Fanuc TP program (LS listing): FM152248.ls

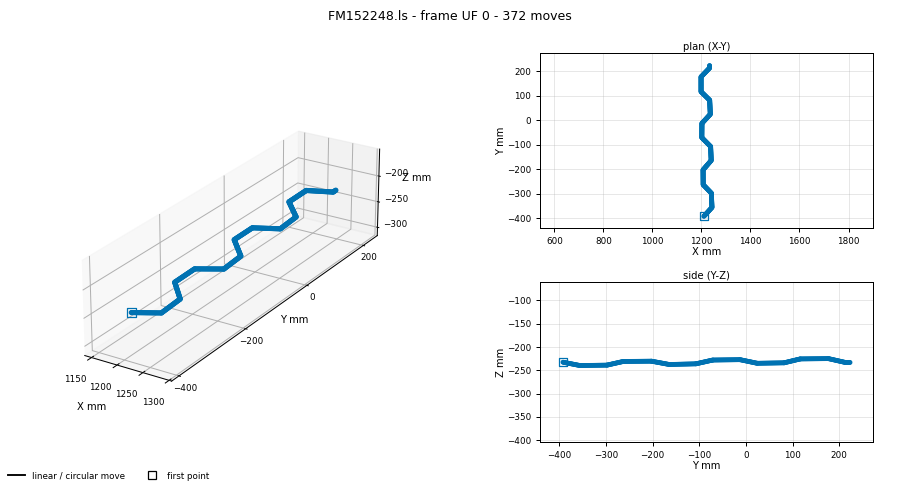
[picture p0: tool path of FM152248.ls in frame UF 0, 372 of 372 moves have a stored position in this frame; points joined in program order, loops and branches not executed]
/PROG  FM152248
/ATTR
OWNER		= MNEDITOR;
COMMENT		= "Auto FANUC move";
PROG_SIZE	= 0;
CREATE		= DATE 26-05-06  TIME 15:22:48;
MODIFIED	= DATE 26-05-06  TIME 15:22:48;
FILE_NAME	= ;
VERSION		= 0;
LINE_COUNT	= 377;
MEMORY_SIZE	= 0;
PROTECT		= READ_WRITE;
TCD:  STACK_SIZE	= 0,
      TASK_PRIORITY	= 50,
      TIME_SLICE	= 0,
      BUSY_LAMP_OFF	= 0,
      ABORT_REQUEST	= 0,
      PAUSE_REQUEST	= 0;
DEFAULT_GROUP	= 1,*,*,*,*;
CONTROL_CODE	= 00000000 00000000;
/MN
   1:  UFRAME_NUM=0 ;
   2:  UTOOL_NUM=1 ;
   3:  R[93]=10 ;
   4:  L P[1] 7mm/sec FINE ;
   5:  L P[2] 7mm/sec CNT50 ;
   6:  L P[3] 7mm/sec CNT50 ;
   7:  L P[4] 7mm/sec CNT50 ;
   8:  L P[5] 7mm/sec CNT50 ;
   9:  L P[6] 7mm/sec CNT50 ;
  10:  L P[7] 7mm/sec CNT50 ;
  11:  L P[8] 7mm/sec CNT50 ;
  12:  L P[9] 7mm/sec CNT50 ;
  13:  L P[10] 7mm/sec CNT50 ;
  14:  L P[11] 7mm/sec CNT50 ;
  15:  L P[12] 7mm/sec CNT50 ;
  16:  L P[13] 7mm/sec CNT50 ;
  17:  L P[14] 7mm/sec CNT50 ;
  18:  L P[15] 7mm/sec CNT50 ;
  19:  L P[16] 7mm/sec CNT50 ;
  20:  L P[17] 7mm/sec CNT50 ;
  21:  L P[18] 7mm/sec CNT50 ;
  22:  L P[19] 7mm/sec CNT50 ;
  23:  L P[20] 7mm/sec CNT50 ;
  24:  L P[21] 7mm/sec CNT50 ;
  25:  L P[22] 7mm/sec CNT50 ;
  26:  L P[23] 7mm/sec CNT50 ;
  27:  L P[24] 7mm/sec CNT50 ;
  28:  L P[25] 7mm/sec CNT50 ;
  29:  L P[26] 7mm/sec CNT50 ;
  30:  L P[27] 7mm/sec CNT50 ;
  31:  L P[28] 7mm/sec CNT50 ;
  32:  L P[29] 7mm/sec CNT50 ;
  33:  L P[30] 7mm/sec CNT50 ;
  34:  L P[31] 7mm/sec CNT50 ;
  35:  L P[32] 7mm/sec CNT50 ;
  36:  L P[33] 7mm/sec CNT50 ;
  37:  L P[34] 7mm/sec CNT50 ;
  38:  L P[35] 7mm/sec CNT50 ;
  39:  L P[36] 7mm/sec CNT50 ;
  40:  L P[37] 7mm/sec CNT50 ;
  41:  L P[38] 7mm/sec CNT50 ;
  42:  L P[39] 7mm/sec CNT50 ;
  43:  L P[40] 7mm/sec CNT50 ;
  44:  L P[41] 7mm/sec CNT50 ;
  45:  L P[42] 7mm/sec CNT50 ;
  46:  L P[43] 7mm/sec CNT50 ;
  47:  L P[44] 7mm/sec CNT50 ;
  48:  L P[45] 7mm/sec CNT50 ;
  49:  L P[46] 7mm/sec CNT50 ;
  50:  L P[47] 7mm/sec CNT50 ;
  51:  L P[48] 7mm/sec CNT50 ;
  52:  L P[49] 7mm/sec CNT50 ;
  53:  L P[50] 7mm/sec CNT50 ;
  54:  L P[51] 7mm/sec CNT50 ;
  55:  L P[52] 7mm/sec CNT50 ;
  56:  L P[53] 7mm/sec CNT50 ;
  57:  L P[54] 7mm/sec CNT50 ;
  58:  L P[55] 7mm/sec CNT50 ;
  59:  L P[56] 7mm/sec CNT50 ;
  60:  L P[57] 7mm/sec CNT50 ;
  61:  L P[58] 7mm/sec CNT50 ;
  62:  L P[59] 7mm/sec CNT50 ;
  63:  L P[60] 7mm/sec CNT50 ;
  64:  L P[61] 7mm/sec CNT50 ;
  65:  L P[62] 7mm/sec CNT50 ;
  66:  L P[63] 7mm/sec CNT50 ;
  67:  L P[64] 7mm/sec CNT50 ;
  68:  L P[65] 7mm/sec CNT50 ;
  69:  L P[66] 7mm/sec CNT50 ;
  70:  L P[67] 7mm/sec CNT50 ;
  71:  L P[68] 7mm/sec CNT50 ;
  72:  L P[69] 7mm/sec CNT50 ;
  73:  L P[70] 7mm/sec CNT50 ;
  74:  L P[71] 7mm/sec CNT50 ;
  75:  L P[72] 7mm/sec CNT50 ;
  76:  L P[73] 7mm/sec CNT50 ;
  77:  L P[74] 7mm/sec CNT50 ;
  78:  L P[75] 7mm/sec CNT50 ;
  79:  L P[76] 7mm/sec CNT50 ;
  80:  L P[77] 7mm/sec CNT50 ;
  81:  L P[78] 7mm/sec CNT50 ;
  82:  L P[79] 7mm/sec CNT50 ;
  83:  L P[80] 7mm/sec CNT50 ;
  84:  L P[81] 7mm/sec CNT50 ;
  85:  L P[82] 7mm/sec CNT50 ;
  86:  L P[83] 7mm/sec CNT50 ;
  87:  L P[84] 7mm/sec CNT50 ;
  88:  L P[85] 7mm/sec CNT50 ;
  89:  L P[86] 7mm/sec CNT50 ;
  90:  L P[87] 7mm/sec CNT50 ;
  91:  L P[88] 7mm/sec CNT50 ;
  92:  L P[89] 7mm/sec CNT50 ;
  93:  L P[90] 7mm/sec CNT50 ;
  94:  L P[91] 7mm/sec CNT50 ;
  95:  L P[92] 7mm/sec CNT50 ;
  96:  L P[93] 7mm/sec CNT50 ;
  97:  L P[94] 7mm/sec CNT50 ;
  98:  L P[95] 7mm/sec CNT50 ;
  99:  L P[96] 7mm/sec CNT50 ;
 100:  L P[97] 7mm/sec CNT50 ;
 101:  L P[98] 7mm/sec CNT50 ;
 102:  L P[99] 7mm/sec CNT50 ;
 103:  L P[100] 7mm/sec CNT50 ;
 104:  L P[101] 7mm/sec CNT50 ;
 105:  L P[102] 7mm/sec CNT50 ;
 106:  L P[103] 7mm/sec CNT50 ;
 107:  L P[104] 7mm/sec CNT50 ;
 108:  L P[105] 7mm/sec CNT50 ;
 109:  L P[106] 7mm/sec CNT50 ;
 110:  L P[107] 7mm/sec CNT50 ;
 111:  L P[108] 7mm/sec CNT50 ;
 112:  L P[109] 7mm/sec CNT50 ;
 113:  L P[110] 7mm/sec CNT50 ;
 114:  L P[111] 7mm/sec CNT50 ;
 115:  L P[112] 7mm/sec CNT50 ;
 116:  L P[113] 7mm/sec CNT50 ;
 117:  L P[114] 7mm/sec CNT50 ;
 118:  L P[115] 7mm/sec CNT50 ;
 119:  L P[116] 7mm/sec CNT50 ;
 120:  L P[117] 7mm/sec CNT50 ;
 121:  L P[118] 7mm/sec CNT50 ;
 122:  L P[119] 7mm/sec CNT50 ;
 123:  L P[120] 7mm/sec CNT50 ;
 124:  L P[121] 7mm/sec CNT50 ;
 125:  L P[122] 7mm/sec CNT50 ;
 126:  L P[123] 7mm/sec CNT50 ;
 127:  L P[124] 7mm/sec CNT50 ;
 128:  L P[125] 7mm/sec CNT50 ;
 129:  L P[126] 7mm/sec CNT50 ;
 130:  L P[127] 7mm/sec CNT50 ;
 131:  L P[128] 7mm/sec CNT50 ;
 132:  L P[129] 7mm/sec CNT50 ;
 133:  L P[130] 7mm/sec CNT50 ;
 134:  L P[131] 7mm/sec CNT50 ;
 135:  L P[132] 7mm/sec CNT50 ;
 136:  L P[133] 7mm/sec CNT50 ;
 137:  L P[134] 7mm/sec CNT50 ;
 138:  L P[135] 7mm/sec CNT50 ;
 139:  L P[136] 7mm/sec CNT50 ;
 140:  L P[137] 7mm/sec CNT50 ;
 141:  L P[138] 7mm/sec CNT50 ;
 142:  L P[139] 7mm/sec CNT50 ;
 143:  L P[140] 7mm/sec CNT50 ;
 144:  L P[141] 7mm/sec CNT50 ;
 145:  L P[142] 7mm/sec CNT50 ;
 146:  L P[143] 7mm/sec CNT50 ;
 147:  L P[144] 7mm/sec CNT50 ;
 148:  L P[145] 7mm/sec CNT50 ;
 149:  L P[146] 7mm/sec CNT50 ;
 150:  L P[147] 7mm/sec CNT50 ;
 151:  L P[148] 7mm/sec CNT50 ;
 152:  L P[149] 7mm/sec CNT50 ;
 153:  L P[150] 7mm/sec CNT50 ;
 154:  L P[151] 7mm/sec CNT50 ;
 155:  L P[152] 7mm/sec CNT50 ;
 156:  L P[153] 7mm/sec CNT50 ;
 157:  L P[154] 7mm/sec CNT50 ;
 158:  L P[155] 7mm/sec CNT50 ;
 159:  L P[156] 7mm/sec CNT50 ;
 160:  L P[157] 7mm/sec CNT50 ;
 161:  L P[158] 7mm/sec CNT50 ;
 162:  L P[159] 7mm/sec CNT50 ;
 163:  L P[160] 7mm/sec CNT50 ;
 164:  L P[161] 7mm/sec CNT50 ;
 165:  L P[162] 7mm/sec CNT50 ;
 166:  L P[163] 7mm/sec CNT50 ;
 167:  L P[164] 7mm/sec CNT50 ;
 168:  L P[165] 7mm/sec CNT50 ;
 169:  L P[166] 7mm/sec CNT50 ;
 170:  L P[167] 7mm/sec CNT50 ;
 171:  L P[168] 7mm/sec CNT50 ;
 172:  L P[169] 7mm/sec CNT50 ;
 173:  L P[170] 7mm/sec CNT50 ;
 174:  L P[171] 7mm/sec CNT50 ;
 175:  L P[172] 7mm/sec CNT50 ;
 176:  L P[173] 7mm/sec CNT50 ;
 177:  L P[174] 7mm/sec CNT50 ;
 178:  L P[175] 7mm/sec CNT50 ;
 179:  L P[176] 7mm/sec CNT50 ;
 180:  L P[177] 7mm/sec CNT50 ;
 181:  L P[178] 7mm/sec CNT50 ;
 182:  L P[179] 7mm/sec CNT50 ;
 183:  L P[180] 7mm/sec CNT50 ;
 184:  L P[181] 7mm/sec CNT50 ;
 185:  L P[182] 7mm/sec CNT50 ;
 186:  L P[183] 7mm/sec CNT50 ;
 187:  L P[184] 7mm/sec CNT50 ;
 188:  L P[185] 7mm/sec CNT50 ;
 189:  L P[186] 7mm/sec CNT50 ;
 190:  L P[187] 7mm/sec CNT50 ;
 191:  L P[188] 7mm/sec CNT50 ;
 192:  L P[189] 7mm/sec CNT50 ;
 193:  L P[190] 7mm/sec CNT50 ;
 194:  L P[191] 7mm/sec CNT50 ;
 195:  L P[192] 7mm/sec CNT50 ;
 196:  L P[193] 7mm/sec CNT50 ;
 197:  L P[194] 7mm/sec CNT50 ;
 198:  L P[195] 7mm/sec CNT50 ;
 199:  L P[196] 7mm/sec CNT50 ;
 200:  L P[197] 7mm/sec CNT50 ;
 201:  L P[198] 7mm/sec CNT50 ;
 202:  L P[199] 7mm/sec CNT50 ;
 203:  L P[200] 7mm/sec CNT50 ;
 204:  L P[201] 7mm/sec CNT50 ;
 205:  L P[202] 7mm/sec CNT50 ;
 206:  L P[203] 7mm/sec CNT50 ;
 207:  L P[204] 7mm/sec CNT50 ;
 208:  L P[205] 7mm/sec CNT50 ;
 209:  L P[206] 7mm/sec CNT50 ;
 210:  L P[207] 7mm/sec CNT50 ;
 211:  L P[208] 7mm/sec CNT50 ;
 212:  L P[209] 7mm/sec CNT50 ;
 213:  L P[210] 7mm/sec CNT50 ;
 214:  L P[211] 7mm/sec CNT50 ;
 215:  L P[212] 7mm/sec CNT50 ;
 216:  L P[213] 7mm/sec CNT50 ;
 217:  L P[214] 7mm/sec CNT50 ;
 218:  L P[215] 7mm/sec CNT50 ;
 219:  L P[216] 7mm/sec CNT50 ;
 220:  L P[217] 7mm/sec CNT50 ;
 221:  L P[218] 7mm/sec CNT50 ;
 222:  L P[219] 7mm/sec CNT50 ;
 223:  L P[220] 7mm/sec CNT50 ;
 224:  L P[221] 7mm/sec CNT50 ;
 225:  L P[222] 7mm/sec CNT50 ;
 226:  L P[223] 7mm/sec CNT50 ;
 227:  L P[224] 7mm/sec CNT50 ;
 228:  L P[225] 7mm/sec CNT50 ;
 229:  L P[226] 7mm/sec CNT50 ;
 230:  L P[227] 7mm/sec CNT50 ;
 231:  L P[228] 7mm/sec CNT50 ;
 232:  L P[229] 7mm/sec CNT50 ;
 233:  L P[230] 7mm/sec CNT50 ;
 234:  L P[231] 7mm/sec CNT50 ;
 235:  L P[232] 7mm/sec CNT50 ;
 236:  L P[233] 7mm/sec CNT50 ;
 237:  L P[234] 7mm/sec CNT50 ;
 238:  L P[235] 7mm/sec CNT50 ;
 239:  L P[236] 7mm/sec CNT50 ;
 240:  L P[237] 7mm/sec CNT50 ;
 241:  L P[238] 7mm/sec CNT50 ;
 242:  L P[239] 7mm/sec CNT50 ;
 243:  L P[240] 7mm/sec CNT50 ;
 244:  L P[241] 7mm/sec CNT50 ;
 245:  L P[242] 7mm/sec CNT50 ;
 246:  L P[243] 7mm/sec CNT50 ;
 247:  L P[244] 7mm/sec CNT50 ;
 248:  L P[245] 7mm/sec CNT50 ;
 249:  L P[246] 7mm/sec CNT50 ;
 250:  L P[247] 7mm/sec CNT50 ;
 251:  L P[248] 7mm/sec CNT50 ;
 252:  L P[249] 7mm/sec CNT50 ;
 253:  L P[250] 7mm/sec CNT50 ;
 254:  L P[251] 7mm/sec CNT50 ;
 255:  L P[252] 7mm/sec CNT50 ;
 256:  L P[253] 7mm/sec CNT50 ;
 257:  L P[254] 7mm/sec CNT50 ;
 258:  L P[255] 7mm/sec CNT50 ;
 259:  L P[256] 7mm/sec CNT50 ;
 260:  L P[257] 7mm/sec CNT50 ;
 261:  L P[258] 7mm/sec CNT50 ;
 262:  L P[259] 7mm/sec CNT50 ;
 263:  L P[260] 7mm/sec CNT50 ;
 264:  L P[261] 7mm/sec CNT50 ;
 265:  L P[262] 7mm/sec CNT50 ;
 266:  L P[263] 7mm/sec CNT50 ;
 267:  L P[264] 7mm/sec CNT50 ;
 268:  L P[265] 7mm/sec CNT50 ;
 269:  L P[266] 7mm/sec CNT50 ;
 270:  L P[267] 7mm/sec CNT50 ;
 271:  L P[268] 7mm/sec CNT50 ;
 272:  L P[269] 7mm/sec CNT50 ;
 273:  L P[270] 7mm/sec CNT50 ;
 274:  L P[271] 7mm/sec CNT50 ;
 275:  L P[272] 7mm/sec CNT50 ;
 276:  L P[273] 7mm/sec CNT50 ;
 277:  L P[274] 7mm/sec CNT50 ;
 278:  L P[275] 7mm/sec CNT50 ;
 279:  L P[276] 7mm/sec CNT50 ;
 280:  L P[277] 7mm/sec CNT50 ;
 281:  L P[278] 7mm/sec CNT50 ;
 282:  L P[279] 7mm/sec CNT50 ;
 283:  L P[280] 7mm/sec CNT50 ;
 284:  L P[281] 7mm/sec CNT50 ;
 285:  L P[282] 7mm/sec CNT50 ;
 286:  L P[283] 7mm/sec CNT50 ;
 287:  L P[284] 7mm/sec CNT50 ;
 288:  L P[285] 7mm/sec CNT50 ;
 289:  L P[286] 7mm/sec CNT50 ;
 290:  L P[287] 7mm/sec CNT50 ;
 291:  L P[288] 7mm/sec CNT50 ;
 292:  L P[289] 7mm/sec CNT50 ;
 293:  L P[290] 7mm/sec CNT50 ;
 294:  L P[291] 7mm/sec CNT50 ;
 295:  L P[292] 7mm/sec CNT50 ;
 296:  L P[293] 7mm/sec CNT50 ;
 297:  L P[294] 7mm/sec CNT50 ;
 298:  L P[295] 7mm/sec CNT50 ;
 299:  L P[296] 7mm/sec CNT50 ;
 300:  L P[297] 7mm/sec CNT50 ;
 301:  L P[298] 7mm/sec CNT50 ;
 302:  L P[299] 7mm/sec CNT50 ;
 303:  L P[300] 7mm/sec CNT50 ;
 304:  L P[301] 7mm/sec CNT50 ;
 305:  L P[302] 7mm/sec CNT50 ;
 306:  L P[303] 7mm/sec CNT50 ;
 307:  L P[304] 7mm/sec CNT50 ;
 308:  L P[305] 7mm/sec CNT50 ;
 309:  L P[306] 7mm/sec CNT50 ;
 310:  L P[307] 7mm/sec CNT50 ;
 311:  L P[308] 7mm/sec CNT50 ;
 312:  L P[309] 7mm/sec CNT50 ;
 313:  L P[310] 7mm/sec CNT50 ;
 314:  L P[311] 7mm/sec CNT50 ;
 315:  L P[312] 7mm/sec CNT50 ;
 316:  L P[313] 7mm/sec CNT50 ;
 317:  L P[314] 7mm/sec CNT50 ;
 318:  L P[315] 7mm/sec CNT50 ;
 319:  L P[316] 7mm/sec CNT50 ;
 320:  L P[317] 7mm/sec CNT50 ;
 321:  L P[318] 7mm/sec CNT50 ;
 322:  L P[319] 7mm/sec CNT50 ;
 323:  L P[320] 7mm/sec CNT50 ;
 324:  L P[321] 7mm/sec CNT50 ;
 325:  L P[322] 7mm/sec CNT50 ;
 326:  L P[323] 7mm/sec CNT50 ;
 327:  L P[324] 7mm/sec CNT50 ;
 328:  L P[325] 7mm/sec CNT50 ;
 329:  L P[326] 7mm/sec CNT50 ;
 330:  L P[327] 7mm/sec CNT50 ;
 331:  L P[328] 7mm/sec CNT50 ;
 332:  L P[329] 7mm/sec CNT50 ;
 333:  L P[330] 7mm/sec CNT50 ;
 334:  L P[331] 7mm/sec CNT50 ;
 335:  L P[332] 7mm/sec CNT50 ;
 336:  L P[333] 7mm/sec CNT50 ;
 337:  L P[334] 7mm/sec CNT50 ;
 338:  L P[335] 7mm/sec CNT50 ;
 339:  L P[336] 7mm/sec CNT50 ;
 340:  L P[337] 7mm/sec CNT50 ;
 341:  L P[338] 7mm/sec CNT50 ;
 342:  L P[339] 7mm/sec CNT50 ;
 343:  L P[340] 7mm/sec CNT50 ;
 344:  L P[341] 7mm/sec CNT50 ;
 345:  L P[342] 7mm/sec CNT50 ;
 346:  L P[343] 7mm/sec CNT50 ;
 347:  L P[344] 7mm/sec CNT50 ;
 348:  L P[345] 7mm/sec CNT50 ;
 349:  L P[346] 7mm/sec CNT50 ;
 350:  L P[347] 7mm/sec CNT50 ;
 351:  L P[348] 7mm/sec CNT50 ;
 352:  L P[349] 7mm/sec CNT50 ;
 353:  L P[350] 7mm/sec CNT50 ;
 354:  L P[351] 7mm/sec CNT50 ;
 355:  L P[352] 7mm/sec CNT50 ;
 356:  L P[353] 7mm/sec CNT50 ;
 357:  L P[354] 7mm/sec CNT50 ;
 358:  L P[355] 7mm/sec CNT50 ;
 359:  L P[356] 7mm/sec CNT50 ;
 360:  L P[357] 7mm/sec CNT50 ;
 361:  L P[358] 7mm/sec CNT50 ;
 362:  L P[359] 7mm/sec CNT50 ;
 363:  L P[360] 7mm/sec CNT50 ;
 364:  L P[361] 7mm/sec CNT50 ;
 365:  L P[362] 7mm/sec CNT50 ;
 366:  L P[363] 7mm/sec CNT50 ;
 367:  L P[364] 7mm/sec CNT50 ;
 368:  L P[365] 7mm/sec CNT50 ;
 369:  L P[366] 7mm/sec CNT50 ;
 370:  L P[367] 7mm/sec CNT50 ;
 371:  L P[368] 7mm/sec CNT50 ;
 372:  L P[369] 7mm/sec CNT50 ;
 373:  L P[370] 7mm/sec CNT50 ;
 374:  L P[371] 7mm/sec CNT50 ;
 375:  L P[372] 7mm/sec FINE ;
 376:  R[93]=1 ;
 377:  END ;
/POS
P[1]{
   GP1:
	UF : 0, UT : 1,		CONFIG : 'N U T, 0, 0, 0',
	X = 1209.863  mm,	Y = -392.091  mm,	Z = -232.573  mm,
	W = 0.000 deg,	P = 30.000 deg,	R = 160.000 deg
};
P[2]{
   GP1:
	UF : 0, UT : 1,		CONFIG : 'N U T, 0, 0, 0',
	X = 1211.194  mm,	Y = -390.625  mm,	Z = -232.860  mm,
	W = 0.000 deg,	P = 30.000 deg,	R = 160.000 deg
};
P[3]{
   GP1:
	UF : 0, UT : 1,		CONFIG : 'N U T, 0, 0, 0',
	X = 1212.524  mm,	Y = -389.159  mm,	Z = -233.146  mm,
	W = 0.000 deg,	P = 30.000 deg,	R = 160.000 deg
};
P[4]{
   GP1:
	UF : 0, UT : 1,		CONFIG : 'N U T, 0, 0, 0',
	X = 1213.854  mm,	Y = -387.693  mm,	Z = -233.432  mm,
	W = 0.000 deg,	P = 30.000 deg,	R = 160.000 deg
};
P[5]{
   GP1:
	UF : 0, UT : 1,		CONFIG : 'N U T, 0, 0, 0',
	X = 1215.184  mm,	Y = -386.228  mm,	Z = -233.719  mm,
	W = 0.000 deg,	P = 30.000 deg,	R = 160.000 deg
};
P[6]{
   GP1:
	UF : 0, UT : 1,		CONFIG : 'N U T, 0, 0, 0',
	X = 1216.515  mm,	Y = -384.762  mm,	Z = -234.005  mm,
	W = 0.000 deg,	P = 30.000 deg,	R = 160.000 deg
};
P[7]{
   GP1:
	UF : 0, UT : 1,		CONFIG : 'N U T, 0, 0, 0',
	X = 1217.845  mm,	Y = -383.296  mm,	Z = -234.291  mm,
	W = 0.000 deg,	P = 30.000 deg,	R = 160.000 deg
};
P[8]{
   GP1:
	UF : 0, UT : 1,		CONFIG : 'N U T, 0, 0, 0',
	X = 1219.175  mm,	Y = -381.830  mm,	Z = -234.578  mm,
	W = 0.000 deg,	P = 30.000 deg,	R = 160.000 deg
};
P[9]{
   GP1:
	UF : 0, UT : 1,		CONFIG : 'N U T, 0, 0, 0',
	X = 1220.505  mm,	Y = -380.365  mm,	Z = -234.864  mm,
	W = 0.000 deg,	P = 30.000 deg,	R = 160.000 deg
};
P[10]{
   GP1:
	UF : 0, UT : 1,		CONFIG : 'N U T, 0, 0, 0',
	X = 1221.836  mm,	Y = -378.899  mm,	Z = -235.150  mm,
	W = 0.000 deg,	P = 30.000 deg,	R = 160.000 deg
};
P[11]{
   GP1:
	UF : 0, UT : 1,		CONFIG : 'N U T, 0, 0, 0',
	X = 1223.166  mm,	Y = -377.433  mm,	Z = -235.437  mm,
	W = 0.000 deg,	P = 30.000 deg,	R = 160.000 deg
};
P[12]{
   GP1:
	UF : 0, UT : 1,		CONFIG : 'N U T, 0, 0, 0',
	X = 1224.496  mm,	Y = -375.967  mm,	Z = -235.723  mm,
	W = 0.000 deg,	P = 30.000 deg,	R = 160.000 deg
};
P[13]{
   GP1:
	UF : 0, UT : 1,		CONFIG : 'N U T, 0, 0, 0',
	X = 1225.826  mm,	Y = -374.502  mm,	Z = -236.010  mm,
	W = 0.000 deg,	P = 30.000 deg,	R = 160.000 deg
};
P[14]{
   GP1:
	UF : 0, UT : 1,		CONFIG : 'N U T, 0, 0, 0',
	X = 1227.157  mm,	Y = -373.036  mm,	Z = -236.296  mm,
	W = 0.000 deg,	P = 30.000 deg,	R = 160.000 deg
};
P[15]{
   GP1:
	UF : 0, UT : 1,		CONFIG : 'N U T, 0, 0, 0',
	X = 1228.487  mm,	Y = -371.570  mm,	Z = -236.582  mm,
	W = 0.000 deg,	P = 30.000 deg,	R = 160.000 deg
};
P[16]{
   GP1:
	UF : 0, UT : 1,		CONFIG : 'N U T, 0, 0, 0',
	X = 1229.817  mm,	Y = -370.104  mm,	Z = -236.869  mm,
	W = 0.000 deg,	P = 30.000 deg,	R = 160.000 deg
};
P[17]{
   GP1:
	UF : 0, UT : 1,		CONFIG : 'N U T, 0, 0, 0',
	X = 1231.147  mm,	Y = -368.639  mm,	Z = -237.155  mm,
	W = 0.000 deg,	P = 30.000 deg,	R = 160.000 deg
};
P[18]{
   GP1:
	UF : 0, UT : 1,		CONFIG : 'N U T, 0, 0, 0',
	X = 1232.478  mm,	Y = -367.173  mm,	Z = -237.441  mm,
	W = 0.000 deg,	P = 30.000 deg,	R = 160.000 deg
};
P[19]{
   GP1:
	UF : 0, UT : 1,		CONFIG : 'N U T, 0, 0, 0',
	X = 1233.808  mm,	Y = -365.707  mm,	Z = -237.728  mm,
	W = 0.000 deg,	P = 30.000 deg,	R = 160.000 deg
};
P[20]{
   GP1:
	UF : 0, UT : 1,		CONFIG : 'N U T, 0, 0, 0',
	X = 1235.138  mm,	Y = -364.241  mm,	Z = -238.014  mm,
	W = 0.000 deg,	P = 30.000 deg,	R = 160.000 deg
};
P[21]{
   GP1:
	UF : 0, UT : 1,		CONFIG : 'N U T, 0, 0, 0',
	X = 1236.468  mm,	Y = -362.776  mm,	Z = -238.300  mm,
	W = 0.000 deg,	P = 30.000 deg,	R = 164.441 deg
};
P[22]{
   GP1:
	UF : 0, UT : 1,		CONFIG : 'N U T, 0, 0, 0',
	X = 1237.799  mm,	Y = -361.310  mm,	Z = -238.587  mm,
	W = 0.000 deg,	P = 30.000 deg,	R = 168.883 deg
};
P[23]{
   GP1:
	UF : 0, UT : 1,		CONFIG : 'N U T, 0, 0, 0',
	X = 1239.129  mm,	Y = -359.844  mm,	Z = -238.873  mm,
	W = 0.000 deg,	P = 30.000 deg,	R = 173.324 deg
};
P[24]{
   GP1:
	UF : 0, UT : 1,		CONFIG : 'N U T, 0, 0, 0',
	X = 1240.459  mm,	Y = -358.378  mm,	Z = -239.159  mm,
	W = 0.000 deg,	P = 30.000 deg,	R = 177.765 deg
};
P[25]{
   GP1:
	UF : 0, UT : 1,		CONFIG : 'N U T, 0, 0, 0',
	X = 1241.789  mm,	Y = -356.912  mm,	Z = -239.446  mm,
	W = 0.000 deg,	P = 30.000 deg,	R = -177.793 deg
};
P[26]{
   GP1:
	UF : 0, UT : 1,		CONFIG : 'N U T, 0, 0, 0',
	X = 1242.946  mm,	Y = -355.638  mm,	Z = -239.695  mm,
	W = 0.000 deg,	P = 30.000 deg,	R = -177.793 deg
};
P[27]{
   GP1:
	UF : 0, UT : 1,		CONFIG : 'N U T, 0, 0, 0',
	X = 1242.936  mm,	Y = -355.377  mm,	Z = -239.691  mm,
	W = 0.000 deg,	P = 30.000 deg,	R = -177.793 deg
};
P[28]{
   GP1:
	UF : 0, UT : 1,		CONFIG : 'N U T, 0, 0, 0',
	X = 1242.859  mm,	Y = -353.379  mm,	Z = -239.662  mm,
	W = 0.000 deg,	P = 30.000 deg,	R = -177.793 deg
};
P[29]{
   GP1:
	UF : 0, UT : 1,		CONFIG : 'N U T, 0, 0, 0',
	X = 1242.782  mm,	Y = -351.381  mm,	Z = -239.633  mm,
	W = 0.000 deg,	P = 30.000 deg,	R = -177.793 deg
};
P[30]{
   GP1:
	UF : 0, UT : 1,		CONFIG : 'N U T, 0, 0, 0',
	X = 1242.705  mm,	Y = -349.382  mm,	Z = -239.604  mm,
	W = 0.000 deg,	P = 30.000 deg,	R = -177.793 deg
};
P[31]{
   GP1:
	UF : 0, UT : 1,		CONFIG : 'N U T, 0, 0, 0',
	X = 1242.628  mm,	Y = -347.384  mm,	Z = -239.575  mm,
	W = 0.000 deg,	P = 30.000 deg,	R = -177.793 deg
};
P[32]{
   GP1:
	UF : 0, UT : 1,		CONFIG : 'N U T, 0, 0, 0',
	X = 1242.551  mm,	Y = -345.386  mm,	Z = -239.546  mm,
	W = 0.000 deg,	P = 30.000 deg,	R = -177.793 deg
};
P[33]{
   GP1:
	UF : 0, UT : 1,		CONFIG : 'N U T, 0, 0, 0',
	X = 1242.474  mm,	Y = -343.388  mm,	Z = -239.517  mm,
	W = 0.000 deg,	P = 30.000 deg,	R = -177.793 deg
};
P[34]{
   GP1:
	UF : 0, UT : 1,		CONFIG : 'N U T, 0, 0, 0',
	X = 1242.397  mm,	Y = -341.389  mm,	Z = -239.488  mm,
	W = 0.000 deg,	P = 30.000 deg,	R = -177.793 deg
};
P[35]{
   GP1:
	UF : 0, UT : 1,		CONFIG : 'N U T, 0, 0, 0',
	X = 1242.320  mm,	Y = -339.391  mm,	Z = -239.459  mm,
	W = 0.000 deg,	P = 30.000 deg,	R = -177.793 deg
};
P[36]{
   GP1:
	UF : 0, UT : 1,		CONFIG : 'N U T, 0, 0, 0',
	X = 1242.243  mm,	Y = -337.393  mm,	Z = -239.430  mm,
	W = 0.000 deg,	P = 30.000 deg,	R = -177.793 deg
};
P[37]{
   GP1:
	UF : 0, UT : 1,		CONFIG : 'N U T, 0, 0, 0',
	X = 1242.166  mm,	Y = -335.394  mm,	Z = -239.401  mm,
	W = 0.000 deg,	P = 30.000 deg,	R = -177.793 deg
};
P[38]{
   GP1:
	UF : 0, UT : 1,		CONFIG : 'N U T, 0, 0, 0',
	X = 1242.089  mm,	Y = -333.396  mm,	Z = -239.372  mm,
	W = 0.000 deg,	P = 30.000 deg,	R = -177.793 deg
};
P[39]{
   GP1:
	UF : 0, UT : 1,		CONFIG : 'N U T, 0, 0, 0',
	X = 1242.012  mm,	Y = -331.398  mm,	Z = -239.342  mm,
	W = 0.000 deg,	P = 30.000 deg,	R = -177.793 deg
};
P[40]{
   GP1:
	UF : 0, UT : 1,		CONFIG : 'N U T, 0, 0, 0',
	X = 1241.935  mm,	Y = -329.399  mm,	Z = -239.313  mm,
	W = 0.000 deg,	P = 30.000 deg,	R = -177.793 deg
};
P[41]{
   GP1:
	UF : 0, UT : 1,		CONFIG : 'N U T, 0, 0, 0',
	X = 1241.858  mm,	Y = -327.401  mm,	Z = -239.284  mm,
	W = 0.000 deg,	P = 30.000 deg,	R = -177.793 deg
};
P[42]{
   GP1:
	UF : 0, UT : 1,		CONFIG : 'N U T, 0, 0, 0',
	X = 1241.781  mm,	Y = -325.403  mm,	Z = -239.255  mm,
	W = 0.000 deg,	P = 30.000 deg,	R = -177.793 deg
};
P[43]{
   GP1:
	UF : 0, UT : 1,		CONFIG : 'N U T, 0, 0, 0',
	X = 1241.704  mm,	Y = -323.405  mm,	Z = -239.226  mm,
	W = 0.000 deg,	P = 30.000 deg,	R = -177.793 deg
};
P[44]{
   GP1:
	UF : 0, UT : 1,		CONFIG : 'N U T, 0, 0, 0',
	X = 1241.627  mm,	Y = -321.406  mm,	Z = -239.197  mm,
	W = 0.000 deg,	P = 30.000 deg,	R = -177.793 deg
};
P[45]{
   GP1:
	UF : 0, UT : 1,		CONFIG : 'N U T, 0, 0, 0',
	X = 1241.550  mm,	Y = -319.408  mm,	Z = -239.168  mm,
	W = 0.000 deg,	P = 30.000 deg,	R = -177.793 deg
};
P[46]{
   GP1:
	UF : 0, UT : 1,		CONFIG : 'N U T, 0, 0, 0',
	X = 1241.473  mm,	Y = -317.410  mm,	Z = -239.139  mm,
	W = 0.000 deg,	P = 30.000 deg,	R = -177.793 deg
};
P[47]{
   GP1:
	UF : 0, UT : 1,		CONFIG : 'N U T, 0, 0, 0',
	X = 1241.396  mm,	Y = -315.411  mm,	Z = -239.110  mm,
	W = 0.000 deg,	P = 30.000 deg,	R = -177.793 deg
};
P[48]{
   GP1:
	UF : 0, UT : 1,		CONFIG : 'N U T, 0, 0, 0',
	X = 1241.319  mm,	Y = -313.413  mm,	Z = -239.081  mm,
	W = 0.000 deg,	P = 30.000 deg,	R = -177.793 deg
};
P[49]{
   GP1:
	UF : 0, UT : 1,		CONFIG : 'N U T, 0, 0, 0',
	X = 1241.242  mm,	Y = -311.415  mm,	Z = -239.052  mm,
	W = 0.000 deg,	P = 30.000 deg,	R = -177.793 deg
};
P[50]{
   GP1:
	UF : 0, UT : 1,		CONFIG : 'N U T, 0, 0, 0',
	X = 1241.165  mm,	Y = -309.416  mm,	Z = -239.023  mm,
	W = 0.000 deg,	P = 30.000 deg,	R = -177.330 deg
};
P[51]{
   GP1:
	UF : 0, UT : 1,		CONFIG : 'N U T, 0, 0, 0',
	X = 1241.088  mm,	Y = -307.418  mm,	Z = -238.994  mm,
	W = 0.000 deg,	P = 30.000 deg,	R = -173.771 deg
};
P[52]{
   GP1:
	UF : 0, UT : 1,		CONFIG : 'N U T, 0, 0, 0',
	X = 1241.011  mm,	Y = -305.420  mm,	Z = -238.965  mm,
	W = 0.000 deg,	P = 30.000 deg,	R = -170.213 deg
};
P[53]{
   GP1:
	UF : 0, UT : 1,		CONFIG : 'N U T, 0, 0, 0',
	X = 1240.934  mm,	Y = -303.421  mm,	Z = -238.936  mm,
	W = 0.000 deg,	P = 30.000 deg,	R = -166.654 deg
};
P[54]{
   GP1:
	UF : 0, UT : 1,		CONFIG : 'N U T, 0, 0, 0',
	X = 1240.857  mm,	Y = -301.423  mm,	Z = -238.907  mm,
	W = 0.000 deg,	P = 30.000 deg,	R = -163.095 deg
};
P[55]{
   GP1:
	UF : 0, UT : 1,		CONFIG : 'N U T, 0, 0, 0',
	X = 1240.780  mm,	Y = -299.425  mm,	Z = -238.878  mm,
	W = 0.000 deg,	P = 30.000 deg,	R = -160.000 deg
};
P[56]{
   GP1:
	UF : 0, UT : 1,		CONFIG : 'N U T, 0, 0, 0',
	X = 1240.717  mm,	Y = -297.777  mm,	Z = -238.854  mm,
	W = 0.000 deg,	P = 30.000 deg,	R = -160.000 deg
};
P[57]{
   GP1:
	UF : 0, UT : 1,		CONFIG : 'N U T, 0, 0, 0',
	X = 1240.477  mm,	Y = -297.528  mm,	Z = -238.798  mm,
	W = 0.000 deg,	P = 30.000 deg,	R = -160.000 deg
};
P[58]{
   GP1:
	UF : 0, UT : 1,		CONFIG : 'N U T, 0, 0, 0',
	X = 1239.108  mm,	Y = -296.105  mm,	Z = -238.477  mm,
	W = 0.000 deg,	P = 30.000 deg,	R = -160.000 deg
};
P[59]{
   GP1:
	UF : 0, UT : 1,		CONFIG : 'N U T, 0, 0, 0',
	X = 1237.740  mm,	Y = -294.682  mm,	Z = -238.157  mm,
	W = 0.000 deg,	P = 30.000 deg,	R = -160.000 deg
};
P[60]{
   GP1:
	UF : 0, UT : 1,		CONFIG : 'N U T, 0, 0, 0',
	X = 1236.371  mm,	Y = -293.259  mm,	Z = -237.836  mm,
	W = 0.000 deg,	P = 30.000 deg,	R = -160.000 deg
};
P[61]{
   GP1:
	UF : 0, UT : 1,		CONFIG : 'N U T, 0, 0, 0',
	X = 1235.003  mm,	Y = -291.836  mm,	Z = -237.516  mm,
	W = 0.000 deg,	P = 30.000 deg,	R = -160.000 deg
};
P[62]{
   GP1:
	UF : 0, UT : 1,		CONFIG : 'N U T, 0, 0, 0',
	X = 1233.634  mm,	Y = -290.413  mm,	Z = -237.196  mm,
	W = 0.000 deg,	P = 30.000 deg,	R = -160.000 deg
};
P[63]{
   GP1:
	UF : 0, UT : 1,		CONFIG : 'N U T, 0, 0, 0',
	X = 1232.265  mm,	Y = -288.990  mm,	Z = -236.875  mm,
	W = 0.000 deg,	P = 30.000 deg,	R = -160.000 deg
};
P[64]{
   GP1:
	UF : 0, UT : 1,		CONFIG : 'N U T, 0, 0, 0',
	X = 1230.897  mm,	Y = -287.568  mm,	Z = -236.555  mm,
	W = 0.000 deg,	P = 30.000 deg,	R = -160.000 deg
};
P[65]{
   GP1:
	UF : 0, UT : 1,		CONFIG : 'N U T, 0, 0, 0',
	X = 1229.528  mm,	Y = -286.145  mm,	Z = -236.234  mm,
	W = 0.000 deg,	P = 30.000 deg,	R = -160.000 deg
};
P[66]{
   GP1:
	UF : 0, UT : 1,		CONFIG : 'N U T, 0, 0, 0',
	X = 1228.160  mm,	Y = -284.722  mm,	Z = -235.914  mm,
	W = 0.000 deg,	P = 30.000 deg,	R = -160.000 deg
};
P[67]{
   GP1:
	UF : 0, UT : 1,		CONFIG : 'N U T, 0, 0, 0',
	X = 1226.791  mm,	Y = -283.299  mm,	Z = -235.594  mm,
	W = 0.000 deg,	P = 30.000 deg,	R = -160.000 deg
};
P[68]{
   GP1:
	UF : 0, UT : 1,		CONFIG : 'N U T, 0, 0, 0',
	X = 1225.423  mm,	Y = -281.876  mm,	Z = -235.273  mm,
	W = 0.000 deg,	P = 30.000 deg,	R = -160.000 deg
};
P[69]{
   GP1:
	UF : 0, UT : 1,		CONFIG : 'N U T, 0, 0, 0',
	X = 1224.054  mm,	Y = -280.453  mm,	Z = -234.953  mm,
	W = 0.000 deg,	P = 30.000 deg,	R = -160.000 deg
};
P[70]{
   GP1:
	UF : 0, UT : 1,		CONFIG : 'N U T, 0, 0, 0',
	X = 1222.686  mm,	Y = -279.031  mm,	Z = -234.632  mm,
	W = 0.000 deg,	P = 30.000 deg,	R = -160.000 deg
};
P[71]{
   GP1:
	UF : 0, UT : 1,		CONFIG : 'N U T, 0, 0, 0',
	X = 1221.317  mm,	Y = -277.608  mm,	Z = -234.312  mm,
	W = 0.000 deg,	P = 30.000 deg,	R = -160.000 deg
};
P[72]{
   GP1:
	UF : 0, UT : 1,		CONFIG : 'N U T, 0, 0, 0',
	X = 1219.949  mm,	Y = -276.185  mm,	Z = -233.992  mm,
	W = 0.000 deg,	P = 30.000 deg,	R = -160.000 deg
};
P[73]{
   GP1:
	UF : 0, UT : 1,		CONFIG : 'N U T, 0, 0, 0',
	X = 1218.580  mm,	Y = -274.762  mm,	Z = -233.671  mm,
	W = 0.000 deg,	P = 30.000 deg,	R = -160.000 deg
};
P[74]{
   GP1:
	UF : 0, UT : 1,		CONFIG : 'N U T, 0, 0, 0',
	X = 1217.212  mm,	Y = -273.339  mm,	Z = -233.351  mm,
	W = 0.000 deg,	P = 30.000 deg,	R = -160.000 deg
};
P[75]{
   GP1:
	UF : 0, UT : 1,		CONFIG : 'N U T, 0, 0, 0',
	X = 1215.843  mm,	Y = -271.916  mm,	Z = -233.030  mm,
	W = 0.000 deg,	P = 30.000 deg,	R = -160.000 deg
};
P[76]{
   GP1:
	UF : 0, UT : 1,		CONFIG : 'N U T, 0, 0, 0',
	X = 1214.475  mm,	Y = -270.494  mm,	Z = -232.710  mm,
	W = 0.000 deg,	P = 30.000 deg,	R = -160.688 deg
};
P[77]{
   GP1:
	UF : 0, UT : 1,		CONFIG : 'N U T, 0, 0, 0',
	X = 1213.106  mm,	Y = -269.071  mm,	Z = -232.390  mm,
	W = 0.000 deg,	P = 30.000 deg,	R = -164.612 deg
};
P[78]{
   GP1:
	UF : 0, UT : 1,		CONFIG : 'N U T, 0, 0, 0',
	X = 1211.738  mm,	Y = -267.648  mm,	Z = -232.069  mm,
	W = 0.000 deg,	P = 30.000 deg,	R = -168.535 deg
};
P[79]{
   GP1:
	UF : 0, UT : 1,		CONFIG : 'N U T, 0, 0, 0',
	X = 1210.369  mm,	Y = -266.225  mm,	Z = -231.749  mm,
	W = 0.000 deg,	P = 30.000 deg,	R = -172.458 deg
};
P[80]{
   GP1:
	UF : 0, UT : 1,		CONFIG : 'N U T, 0, 0, 0',
	X = 1209.000  mm,	Y = -264.802  mm,	Z = -231.429  mm,
	W = 0.000 deg,	P = 30.000 deg,	R = -176.382 deg
};
P[81]{
   GP1:
	UF : 0, UT : 1,		CONFIG : 'N U T, 0, 0, 0',
	X = 1207.632  mm,	Y = -263.379  mm,	Z = -231.108  mm,
	W = 0.000 deg,	P = 30.000 deg,	R = -179.617 deg
};
P[82]{
   GP1:
	UF : 0, UT : 1,		CONFIG : 'N U T, 0, 0, 0',
	X = 1207.094  mm,	Y = -262.820  mm,	Z = -230.982  mm,
	W = 0.000 deg,	P = 30.000 deg,	R = -179.617 deg
};
P[83]{
   GP1:
	UF : 0, UT : 1,		CONFIG : 'N U T, 0, 0, 0',
	X = 1207.086  mm,	Y = -261.606  mm,	Z = -230.970  mm,
	W = 0.000 deg,	P = 30.000 deg,	R = -179.617 deg
};
P[84]{
   GP1:
	UF : 0, UT : 1,		CONFIG : 'N U T, 0, 0, 0',
	X = 1207.073  mm,	Y = -259.606  mm,	Z = -230.950  mm,
	W = 0.000 deg,	P = 30.000 deg,	R = -179.617 deg
};
P[85]{
   GP1:
	UF : 0, UT : 1,		CONFIG : 'N U T, 0, 0, 0',
	X = 1207.059  mm,	Y = -257.606  mm,	Z = -230.930  mm,
	W = 0.000 deg,	P = 30.000 deg,	R = -179.617 deg
};
P[86]{
   GP1:
	UF : 0, UT : 1,		CONFIG : 'N U T, 0, 0, 0',
	X = 1207.046  mm,	Y = -255.607  mm,	Z = -230.910  mm,
	W = 0.000 deg,	P = 30.000 deg,	R = -179.617 deg
};
P[87]{
   GP1:
	UF : 0, UT : 1,		CONFIG : 'N U T, 0, 0, 0',
	X = 1207.033  mm,	Y = -253.607  mm,	Z = -230.890  mm,
	W = 0.000 deg,	P = 30.000 deg,	R = -179.617 deg
};
P[88]{
   GP1:
	UF : 0, UT : 1,		CONFIG : 'N U T, 0, 0, 0',
	X = 1207.019  mm,	Y = -251.607  mm,	Z = -230.870  mm,
	W = 0.000 deg,	P = 30.000 deg,	R = -179.617 deg
};
P[89]{
   GP1:
	UF : 0, UT : 1,		CONFIG : 'N U T, 0, 0, 0',
	X = 1207.006  mm,	Y = -249.607  mm,	Z = -230.850  mm,
	W = 0.000 deg,	P = 30.000 deg,	R = -179.617 deg
};
P[90]{
   GP1:
	UF : 0, UT : 1,		CONFIG : 'N U T, 0, 0, 0',
	X = 1206.993  mm,	Y = -247.607  mm,	Z = -230.830  mm,
	W = 0.000 deg,	P = 30.000 deg,	R = -179.617 deg
};
P[91]{
   GP1:
	UF : 0, UT : 1,		CONFIG : 'N U T, 0, 0, 0',
	X = 1206.979  mm,	Y = -245.607  mm,	Z = -230.810  mm,
	W = 0.000 deg,	P = 30.000 deg,	R = -179.617 deg
};
P[92]{
   GP1:
	UF : 0, UT : 1,		CONFIG : 'N U T, 0, 0, 0',
	X = 1206.966  mm,	Y = -243.607  mm,	Z = -230.790  mm,
	W = 0.000 deg,	P = 30.000 deg,	R = -179.617 deg
};
P[93]{
   GP1:
	UF : 0, UT : 1,		CONFIG : 'N U T, 0, 0, 0',
	X = 1206.952  mm,	Y = -241.608  mm,	Z = -230.770  mm,
	W = 0.000 deg,	P = 30.000 deg,	R = -179.617 deg
};
P[94]{
   GP1:
	UF : 0, UT : 1,		CONFIG : 'N U T, 0, 0, 0',
	X = 1206.939  mm,	Y = -239.608  mm,	Z = -230.750  mm,
	W = 0.000 deg,	P = 30.000 deg,	R = -179.617 deg
};
P[95]{
   GP1:
	UF : 0, UT : 1,		CONFIG : 'N U T, 0, 0, 0',
	X = 1206.926  mm,	Y = -237.608  mm,	Z = -230.730  mm,
	W = 0.000 deg,	P = 30.000 deg,	R = -179.617 deg
};
P[96]{
   GP1:
	UF : 0, UT : 1,		CONFIG : 'N U T, 0, 0, 0',
	X = 1206.912  mm,	Y = -235.608  mm,	Z = -230.710  mm,
	W = 0.000 deg,	P = 30.000 deg,	R = -179.617 deg
};
P[97]{
   GP1:
	UF : 0, UT : 1,		CONFIG : 'N U T, 0, 0, 0',
	X = 1206.899  mm,	Y = -233.608  mm,	Z = -230.690  mm,
	W = 0.000 deg,	P = 30.000 deg,	R = -179.617 deg
};
P[98]{
   GP1:
	UF : 0, UT : 1,		CONFIG : 'N U T, 0, 0, 0',
	X = 1206.886  mm,	Y = -231.608  mm,	Z = -230.670  mm,
	W = 0.000 deg,	P = 30.000 deg,	R = -179.617 deg
};
P[99]{
   GP1:
	UF : 0, UT : 1,		CONFIG : 'N U T, 0, 0, 0',
	X = 1206.872  mm,	Y = -229.608  mm,	Z = -230.649  mm,
	W = 0.000 deg,	P = 30.000 deg,	R = -179.617 deg
};
P[100]{
   GP1:
	UF : 0, UT : 1,		CONFIG : 'N U T, 0, 0, 0',
	X = 1206.859  mm,	Y = -227.609  mm,	Z = -230.629  mm,
	W = 0.000 deg,	P = 30.000 deg,	R = -179.617 deg
};
P[101]{
   GP1:
	UF : 0, UT : 1,		CONFIG : 'N U T, 0, 0, 0',
	X = 1206.845  mm,	Y = -225.609  mm,	Z = -230.609  mm,
	W = 0.000 deg,	P = 30.000 deg,	R = -179.617 deg
};
P[102]{
   GP1:
	UF : 0, UT : 1,		CONFIG : 'N U T, 0, 0, 0',
	X = 1206.832  mm,	Y = -223.609  mm,	Z = -230.589  mm,
	W = 0.000 deg,	P = 30.000 deg,	R = -179.617 deg
};
P[103]{
   GP1:
	UF : 0, UT : 1,		CONFIG : 'N U T, 0, 0, 0',
	X = 1206.819  mm,	Y = -221.609  mm,	Z = -230.569  mm,
	W = 0.000 deg,	P = 30.000 deg,	R = -179.617 deg
};
P[104]{
   GP1:
	UF : 0, UT : 1,		CONFIG : 'N U T, 0, 0, 0',
	X = 1206.805  mm,	Y = -219.609  mm,	Z = -230.549  mm,
	W = 0.000 deg,	P = 30.000 deg,	R = -179.617 deg
};
P[105]{
   GP1:
	UF : 0, UT : 1,		CONFIG : 'N U T, 0, 0, 0',
	X = 1206.792  mm,	Y = -217.609  mm,	Z = -230.529  mm,
	W = 0.000 deg,	P = 30.000 deg,	R = -179.617 deg
};
P[106]{
   GP1:
	UF : 0, UT : 1,		CONFIG : 'N U T, 0, 0, 0',
	X = 1206.779  mm,	Y = -215.609  mm,	Z = -230.509  mm,
	W = 0.000 deg,	P = 30.000 deg,	R = -179.617 deg
};
P[107]{
   GP1:
	UF : 0, UT : 1,		CONFIG : 'N U T, 0, 0, 0',
	X = 1206.765  mm,	Y = -213.610  mm,	Z = -230.489  mm,
	W = 0.000 deg,	P = 30.000 deg,	R = -179.617 deg
};
P[108]{
   GP1:
	UF : 0, UT : 1,		CONFIG : 'N U T, 0, 0, 0',
	X = 1206.752  mm,	Y = -211.610  mm,	Z = -230.469  mm,
	W = 0.000 deg,	P = 30.000 deg,	R = -179.617 deg
};
P[109]{
   GP1:
	UF : 0, UT : 1,		CONFIG : 'N U T, 0, 0, 0',
	X = 1206.738  mm,	Y = -209.610  mm,	Z = -230.449  mm,
	W = 0.000 deg,	P = 30.000 deg,	R = 173.831 deg
};
P[110]{
   GP1:
	UF : 0, UT : 1,		CONFIG : 'N U T, 0, 0, 0',
	X = 1206.725  mm,	Y = -207.610  mm,	Z = -230.429  mm,
	W = 0.000 deg,	P = 30.000 deg,	R = 169.755 deg
};
P[111]{
   GP1:
	UF : 0, UT : 1,		CONFIG : 'N U T, 0, 0, 0',
	X = 1206.712  mm,	Y = -205.610  mm,	Z = -230.409  mm,
	W = 0.000 deg,	P = 30.000 deg,	R = 165.678 deg
};
P[112]{
   GP1:
	UF : 0, UT : 1,		CONFIG : 'N U T, 0, 0, 0',
	X = 1206.698  mm,	Y = -203.610  mm,	Z = -230.389  mm,
	W = 0.000 deg,	P = 30.000 deg,	R = 161.601 deg
};
P[113]{
   GP1:
	UF : 0, UT : 1,		CONFIG : 'N U T, 0, 0, 0',
	X = 1206.691  mm,	Y = -202.486  mm,	Z = -230.378  mm,
	W = 0.000 deg,	P = 30.000 deg,	R = 160.000 deg
};
P[114]{
   GP1:
	UF : 0, UT : 1,		CONFIG : 'N U T, 0, 0, 0',
	X = 1207.258  mm,	Y = -201.830  mm,	Z = -230.499  mm,
	W = 0.000 deg,	P = 30.000 deg,	R = 160.000 deg
};
P[115]{
   GP1:
	UF : 0, UT : 1,		CONFIG : 'N U T, 0, 0, 0',
	X = 1208.552  mm,	Y = -200.331  mm,	Z = -230.777  mm,
	W = 0.000 deg,	P = 30.000 deg,	R = 160.000 deg
};
P[116]{
   GP1:
	UF : 0, UT : 1,		CONFIG : 'N U T, 0, 0, 0',
	X = 1209.847  mm,	Y = -198.833  mm,	Z = -231.055  mm,
	W = 0.000 deg,	P = 30.000 deg,	R = 160.000 deg
};
P[117]{
   GP1:
	UF : 0, UT : 1,		CONFIG : 'N U T, 0, 0, 0',
	X = 1211.142  mm,	Y = -197.334  mm,	Z = -231.333  mm,
	W = 0.000 deg,	P = 30.000 deg,	R = 160.000 deg
};
P[118]{
   GP1:
	UF : 0, UT : 1,		CONFIG : 'N U T, 0, 0, 0',
	X = 1212.437  mm,	Y = -195.835  mm,	Z = -231.611  mm,
	W = 0.000 deg,	P = 30.000 deg,	R = 160.000 deg
};
P[119]{
   GP1:
	UF : 0, UT : 1,		CONFIG : 'N U T, 0, 0, 0',
	X = 1213.732  mm,	Y = -194.336  mm,	Z = -231.889  mm,
	W = 0.000 deg,	P = 30.000 deg,	R = 160.000 deg
};
P[120]{
   GP1:
	UF : 0, UT : 1,		CONFIG : 'N U T, 0, 0, 0',
	X = 1215.027  mm,	Y = -192.838  mm,	Z = -232.167  mm,
	W = 0.000 deg,	P = 30.000 deg,	R = 160.000 deg
};
P[121]{
   GP1:
	UF : 0, UT : 1,		CONFIG : 'N U T, 0, 0, 0',
	X = 1216.322  mm,	Y = -191.339  mm,	Z = -232.445  mm,
	W = 0.000 deg,	P = 30.000 deg,	R = 160.000 deg
};
P[122]{
   GP1:
	UF : 0, UT : 1,		CONFIG : 'N U T, 0, 0, 0',
	X = 1217.616  mm,	Y = -189.840  mm,	Z = -232.723  mm,
	W = 0.000 deg,	P = 30.000 deg,	R = 160.000 deg
};
P[123]{
   GP1:
	UF : 0, UT : 1,		CONFIG : 'N U T, 0, 0, 0',
	X = 1218.911  mm,	Y = -188.342  mm,	Z = -233.001  mm,
	W = 0.000 deg,	P = 30.000 deg,	R = 160.000 deg
};
P[124]{
   GP1:
	UF : 0, UT : 1,		CONFIG : 'N U T, 0, 0, 0',
	X = 1220.206  mm,	Y = -186.843  mm,	Z = -233.279  mm,
	W = 0.000 deg,	P = 30.000 deg,	R = 160.000 deg
};
P[125]{
   GP1:
	UF : 0, UT : 1,		CONFIG : 'N U T, 0, 0, 0',
	X = 1221.501  mm,	Y = -185.344  mm,	Z = -233.557  mm,
	W = 0.000 deg,	P = 30.000 deg,	R = 160.000 deg
};
P[126]{
   GP1:
	UF : 0, UT : 1,		CONFIG : 'N U T, 0, 0, 0',
	X = 1222.796  mm,	Y = -183.846  mm,	Z = -233.835  mm,
	W = 0.000 deg,	P = 30.000 deg,	R = 160.000 deg
};
P[127]{
   GP1:
	UF : 0, UT : 1,		CONFIG : 'N U T, 0, 0, 0',
	X = 1224.091  mm,	Y = -182.347  mm,	Z = -234.113  mm,
	W = 0.000 deg,	P = 30.000 deg,	R = 160.000 deg
};
P[128]{
   GP1:
	UF : 0, UT : 1,		CONFIG : 'N U T, 0, 0, 0',
	X = 1225.385  mm,	Y = -180.848  mm,	Z = -234.391  mm,
	W = 0.000 deg,	P = 30.000 deg,	R = 160.000 deg
};
P[129]{
   GP1:
	UF : 0, UT : 1,		CONFIG : 'N U T, 0, 0, 0',
	X = 1226.680  mm,	Y = -179.349  mm,	Z = -234.669  mm,
	W = 0.000 deg,	P = 30.000 deg,	R = 160.000 deg
};
P[130]{
   GP1:
	UF : 0, UT : 1,		CONFIG : 'N U T, 0, 0, 0',
	X = 1227.975  mm,	Y = -177.851  mm,	Z = -234.947  mm,
	W = 0.000 deg,	P = 30.000 deg,	R = 160.000 deg
};
P[131]{
   GP1:
	UF : 0, UT : 1,		CONFIG : 'N U T, 0, 0, 0',
	X = 1229.270  mm,	Y = -176.352  mm,	Z = -235.225  mm,
	W = 0.000 deg,	P = 30.000 deg,	R = 160.000 deg
};
P[132]{
   GP1:
	UF : 0, UT : 1,		CONFIG : 'N U T, 0, 0, 0',
	X = 1230.565  mm,	Y = -174.853  mm,	Z = -235.503  mm,
	W = 0.000 deg,	P = 30.000 deg,	R = 160.000 deg
};
P[133]{
   GP1:
	UF : 0, UT : 1,		CONFIG : 'N U T, 0, 0, 0',
	X = 1231.860  mm,	Y = -173.355  mm,	Z = -235.781  mm,
	W = 0.000 deg,	P = 30.000 deg,	R = 160.000 deg
};
P[134]{
   GP1:
	UF : 0, UT : 1,		CONFIG : 'N U T, 0, 0, 0',
	X = 1233.154  mm,	Y = -171.856  mm,	Z = -236.059  mm,
	W = 0.000 deg,	P = 30.000 deg,	R = 160.000 deg
};
P[135]{
   GP1:
	UF : 0, UT : 1,		CONFIG : 'N U T, 0, 0, 0',
	X = 1234.449  mm,	Y = -170.357  mm,	Z = -236.337  mm,
	W = 0.000 deg,	P = 30.000 deg,	R = 166.370 deg
};
P[136]{
   GP1:
	UF : 0, UT : 1,		CONFIG : 'N U T, 0, 0, 0',
	X = 1235.744  mm,	Y = -168.859  mm,	Z = -236.615  mm,
	W = 0.000 deg,	P = 30.000 deg,	R = 170.801 deg
};
P[137]{
   GP1:
	UF : 0, UT : 1,		CONFIG : 'N U T, 0, 0, 0',
	X = 1237.039  mm,	Y = -167.360  mm,	Z = -236.893  mm,
	W = 0.000 deg,	P = 30.000 deg,	R = 175.231 deg
};
P[138]{
   GP1:
	UF : 0, UT : 1,		CONFIG : 'N U T, 0, 0, 0',
	X = 1238.334  mm,	Y = -165.861  mm,	Z = -237.171  mm,
	W = 0.000 deg,	P = 30.000 deg,	R = 179.662 deg
};
P[139]{
   GP1:
	UF : 0, UT : 1,		CONFIG : 'N U T, 0, 0, 0',
	X = 1239.629  mm,	Y = -164.362  mm,	Z = -237.449  mm,
	W = 0.000 deg,	P = 30.000 deg,	R = -177.847 deg
};
P[140]{
   GP1:
	UF : 0, UT : 1,		CONFIG : 'N U T, 0, 0, 0',
	X = 1239.788  mm,	Y = -164.178  mm,	Z = -237.484  mm,
	W = 0.000 deg,	P = 30.000 deg,	R = -177.847 deg
};
P[141]{
   GP1:
	UF : 0, UT : 1,		CONFIG : 'N U T, 0, 0, 0',
	X = 1239.722  mm,	Y = -162.426  mm,	Z = -237.441  mm,
	W = 0.000 deg,	P = 30.000 deg,	R = -177.847 deg
};
P[142]{
   GP1:
	UF : 0, UT : 1,		CONFIG : 'N U T, 0, 0, 0',
	X = 1239.647  mm,	Y = -160.428  mm,	Z = -237.391  mm,
	W = 0.000 deg,	P = 30.000 deg,	R = -177.847 deg
};
P[143]{
   GP1:
	UF : 0, UT : 1,		CONFIG : 'N U T, 0, 0, 0',
	X = 1239.572  mm,	Y = -158.430  mm,	Z = -237.342  mm,
	W = 0.000 deg,	P = 30.000 deg,	R = -177.847 deg
};
P[144]{
   GP1:
	UF : 0, UT : 1,		CONFIG : 'N U T, 0, 0, 0',
	X = 1239.497  mm,	Y = -156.432  mm,	Z = -237.293  mm,
	W = 0.000 deg,	P = 30.000 deg,	R = -177.847 deg
};
P[145]{
   GP1:
	UF : 0, UT : 1,		CONFIG : 'N U T, 0, 0, 0',
	X = 1239.422  mm,	Y = -154.434  mm,	Z = -237.244  mm,
	W = 0.000 deg,	P = 30.000 deg,	R = -177.847 deg
};
P[146]{
   GP1:
	UF : 0, UT : 1,		CONFIG : 'N U T, 0, 0, 0',
	X = 1239.346  mm,	Y = -152.436  mm,	Z = -237.195  mm,
	W = 0.000 deg,	P = 30.000 deg,	R = -177.847 deg
};
P[147]{
   GP1:
	UF : 0, UT : 1,		CONFIG : 'N U T, 0, 0, 0',
	X = 1239.271  mm,	Y = -150.438  mm,	Z = -237.146  mm,
	W = 0.000 deg,	P = 30.000 deg,	R = -177.847 deg
};
P[148]{
   GP1:
	UF : 0, UT : 1,		CONFIG : 'N U T, 0, 0, 0',
	X = 1239.196  mm,	Y = -148.440  mm,	Z = -237.097  mm,
	W = 0.000 deg,	P = 30.000 deg,	R = -177.847 deg
};
P[149]{
   GP1:
	UF : 0, UT : 1,		CONFIG : 'N U T, 0, 0, 0',
	X = 1239.121  mm,	Y = -146.442  mm,	Z = -237.048  mm,
	W = 0.000 deg,	P = 30.000 deg,	R = -177.847 deg
};
P[150]{
   GP1:
	UF : 0, UT : 1,		CONFIG : 'N U T, 0, 0, 0',
	X = 1239.046  mm,	Y = -144.444  mm,	Z = -236.999  mm,
	W = 0.000 deg,	P = 30.000 deg,	R = -177.847 deg
};
P[151]{
   GP1:
	UF : 0, UT : 1,		CONFIG : 'N U T, 0, 0, 0',
	X = 1238.971  mm,	Y = -142.446  mm,	Z = -236.950  mm,
	W = 0.000 deg,	P = 30.000 deg,	R = -177.847 deg
};
P[152]{
   GP1:
	UF : 0, UT : 1,		CONFIG : 'N U T, 0, 0, 0',
	X = 1238.896  mm,	Y = -140.448  mm,	Z = -236.901  mm,
	W = 0.000 deg,	P = 30.000 deg,	R = -177.847 deg
};
P[153]{
   GP1:
	UF : 0, UT : 1,		CONFIG : 'N U T, 0, 0, 0',
	X = 1238.821  mm,	Y = -138.450  mm,	Z = -236.852  mm,
	W = 0.000 deg,	P = 30.000 deg,	R = -177.847 deg
};
P[154]{
   GP1:
	UF : 0, UT : 1,		CONFIG : 'N U T, 0, 0, 0',
	X = 1238.746  mm,	Y = -136.452  mm,	Z = -236.802  mm,
	W = 0.000 deg,	P = 30.000 deg,	R = -177.847 deg
};
P[155]{
   GP1:
	UF : 0, UT : 1,		CONFIG : 'N U T, 0, 0, 0',
	X = 1238.670  mm,	Y = -134.454  mm,	Z = -236.753  mm,
	W = 0.000 deg,	P = 30.000 deg,	R = -177.847 deg
};
P[156]{
   GP1:
	UF : 0, UT : 1,		CONFIG : 'N U T, 0, 0, 0',
	X = 1238.595  mm,	Y = -132.456  mm,	Z = -236.704  mm,
	W = 0.000 deg,	P = 30.000 deg,	R = -177.847 deg
};
P[157]{
   GP1:
	UF : 0, UT : 1,		CONFIG : 'N U T, 0, 0, 0',
	X = 1238.520  mm,	Y = -130.458  mm,	Z = -236.655  mm,
	W = 0.000 deg,	P = 30.000 deg,	R = -177.847 deg
};
P[158]{
   GP1:
	UF : 0, UT : 1,		CONFIG : 'N U T, 0, 0, 0',
	X = 1238.445  mm,	Y = -128.460  mm,	Z = -236.606  mm,
	W = 0.000 deg,	P = 30.000 deg,	R = -177.847 deg
};
P[159]{
   GP1:
	UF : 0, UT : 1,		CONFIG : 'N U T, 0, 0, 0',
	X = 1238.370  mm,	Y = -126.462  mm,	Z = -236.557  mm,
	W = 0.000 deg,	P = 30.000 deg,	R = -177.847 deg
};
P[160]{
   GP1:
	UF : 0, UT : 1,		CONFIG : 'N U T, 0, 0, 0',
	X = 1238.295  mm,	Y = -124.464  mm,	Z = -236.508  mm,
	W = 0.000 deg,	P = 30.000 deg,	R = -177.847 deg
};
P[161]{
   GP1:
	UF : 0, UT : 1,		CONFIG : 'N U T, 0, 0, 0',
	X = 1238.220  mm,	Y = -122.466  mm,	Z = -236.459  mm,
	W = 0.000 deg,	P = 30.000 deg,	R = -177.847 deg
};
P[162]{
   GP1:
	UF : 0, UT : 1,		CONFIG : 'N U T, 0, 0, 0',
	X = 1238.145  mm,	Y = -120.468  mm,	Z = -236.410  mm,
	W = 0.000 deg,	P = 30.000 deg,	R = -177.847 deg
};
P[163]{
   GP1:
	UF : 0, UT : 1,		CONFIG : 'N U T, 0, 0, 0',
	X = 1238.070  mm,	Y = -118.470  mm,	Z = -236.361  mm,
	W = 0.000 deg,	P = 30.000 deg,	R = -177.847 deg
};
P[164]{
   GP1:
	UF : 0, UT : 1,		CONFIG : 'N U T, 0, 0, 0',
	X = 1237.994  mm,	Y = -116.472  mm,	Z = -236.312  mm,
	W = 0.000 deg,	P = 30.000 deg,	R = -177.847 deg
};
P[165]{
   GP1:
	UF : 0, UT : 1,		CONFIG : 'N U T, 0, 0, 0',
	X = 1237.919  mm,	Y = -114.474  mm,	Z = -236.262  mm,
	W = 0.000 deg,	P = 30.000 deg,	R = -171.147 deg
};
P[166]{
   GP1:
	UF : 0, UT : 1,		CONFIG : 'N U T, 0, 0, 0',
	X = 1237.844  mm,	Y = -112.476  mm,	Z = -236.213  mm,
	W = 0.000 deg,	P = 30.000 deg,	R = -167.577 deg
};
P[167]{
   GP1:
	UF : 0, UT : 1,		CONFIG : 'N U T, 0, 0, 0',
	X = 1237.769  mm,	Y = -110.478  mm,	Z = -236.164  mm,
	W = 0.000 deg,	P = 30.000 deg,	R = -164.008 deg
};
P[168]{
   GP1:
	UF : 0, UT : 1,		CONFIG : 'N U T, 0, 0, 0',
	X = 1237.694  mm,	Y = -108.480  mm,	Z = -236.115  mm,
	W = 0.000 deg,	P = 30.000 deg,	R = -160.439 deg
};
P[169]{
   GP1:
	UF : 0, UT : 1,		CONFIG : 'N U T, 0, 0, 0',
	X = 1237.653  mm,	Y = -107.383  mm,	Z = -236.088  mm,
	W = 0.000 deg,	P = 30.000 deg,	R = -160.000 deg
};
P[170]{
   GP1:
	UF : 0, UT : 1,		CONFIG : 'N U T, 0, 0, 0',
	X = 1237.027  mm,	Y = -106.750  mm,	Z = -235.947  mm,
	W = 0.000 deg,	P = 30.000 deg,	R = -160.000 deg
};
P[171]{
   GP1:
	UF : 0, UT : 1,		CONFIG : 'N U T, 0, 0, 0',
	X = 1235.638  mm,	Y = -105.346  mm,	Z = -235.632  mm,
	W = 0.000 deg,	P = 30.000 deg,	R = -160.000 deg
};
P[172]{
   GP1:
	UF : 0, UT : 1,		CONFIG : 'N U T, 0, 0, 0',
	X = 1234.249  mm,	Y = -103.941  mm,	Z = -235.318  mm,
	W = 0.000 deg,	P = 30.000 deg,	R = -160.000 deg
};
P[173]{
   GP1:
	UF : 0, UT : 1,		CONFIG : 'N U T, 0, 0, 0',
	X = 1232.860  mm,	Y = -102.537  mm,	Z = -235.004  mm,
	W = 0.000 deg,	P = 30.000 deg,	R = -160.000 deg
};
P[174]{
   GP1:
	UF : 0, UT : 1,		CONFIG : 'N U T, 0, 0, 0',
	X = 1231.471  mm,	Y = -101.133  mm,	Z = -234.690  mm,
	W = 0.000 deg,	P = 30.000 deg,	R = -160.000 deg
};
P[175]{
   GP1:
	UF : 0, UT : 1,		CONFIG : 'N U T, 0, 0, 0',
	X = 1230.082  mm,	Y = -99.728  mm,	Z = -234.376  mm,
	W = 0.000 deg,	P = 30.000 deg,	R = -160.000 deg
};
P[176]{
   GP1:
	UF : 0, UT : 1,		CONFIG : 'N U T, 0, 0, 0',
	X = 1228.693  mm,	Y = -98.324  mm,	Z = -234.062  mm,
	W = 0.000 deg,	P = 30.000 deg,	R = -160.000 deg
};
P[177]{
   GP1:
	UF : 0, UT : 1,		CONFIG : 'N U T, 0, 0, 0',
	X = 1227.304  mm,	Y = -96.920  mm,	Z = -233.747  mm,
	W = 0.000 deg,	P = 30.000 deg,	R = -160.000 deg
};
P[178]{
   GP1:
	UF : 0, UT : 1,		CONFIG : 'N U T, 0, 0, 0',
	X = 1225.915  mm,	Y = -95.516  mm,	Z = -233.433  mm,
	W = 0.000 deg,	P = 30.000 deg,	R = -160.000 deg
};
P[179]{
   GP1:
	UF : 0, UT : 1,		CONFIG : 'N U T, 0, 0, 0',
	X = 1224.526  mm,	Y = -94.111  mm,	Z = -233.119  mm,
	W = 0.000 deg,	P = 30.000 deg,	R = -160.000 deg
};
P[180]{
   GP1:
	UF : 0, UT : 1,		CONFIG : 'N U T, 0, 0, 0',
	X = 1223.137  mm,	Y = -92.707  mm,	Z = -232.805  mm,
	W = 0.000 deg,	P = 30.000 deg,	R = -160.000 deg
};
P[181]{
   GP1:
	UF : 0, UT : 1,		CONFIG : 'N U T, 0, 0, 0',
	X = 1221.748  mm,	Y = -91.303  mm,	Z = -232.491  mm,
	W = 0.000 deg,	P = 30.000 deg,	R = -160.000 deg
};
P[182]{
   GP1:
	UF : 0, UT : 1,		CONFIG : 'N U T, 0, 0, 0',
	X = 1220.359  mm,	Y = -89.899  mm,	Z = -232.177  mm,
	W = 0.000 deg,	P = 30.000 deg,	R = -160.000 deg
};
P[183]{
   GP1:
	UF : 0, UT : 1,		CONFIG : 'N U T, 0, 0, 0',
	X = 1218.970  mm,	Y = -88.494  mm,	Z = -231.862  mm,
	W = 0.000 deg,	P = 30.000 deg,	R = -160.000 deg
};
P[184]{
   GP1:
	UF : 0, UT : 1,		CONFIG : 'N U T, 0, 0, 0',
	X = 1217.581  mm,	Y = -87.090  mm,	Z = -231.548  mm,
	W = 0.000 deg,	P = 30.000 deg,	R = -160.000 deg
};
P[185]{
   GP1:
	UF : 0, UT : 1,		CONFIG : 'N U T, 0, 0, 0',
	X = 1216.192  mm,	Y = -85.686  mm,	Z = -231.234  mm,
	W = 0.000 deg,	P = 30.000 deg,	R = -160.000 deg
};
P[186]{
   GP1:
	UF : 0, UT : 1,		CONFIG : 'N U T, 0, 0, 0',
	X = 1214.803  mm,	Y = -84.281  mm,	Z = -230.920  mm,
	W = 0.000 deg,	P = 30.000 deg,	R = -160.000 deg
};
P[187]{
   GP1:
	UF : 0, UT : 1,		CONFIG : 'N U T, 0, 0, 0',
	X = 1213.414  mm,	Y = -82.877  mm,	Z = -230.606  mm,
	W = 0.000 deg,	P = 30.000 deg,	R = -160.000 deg
};
P[188]{
   GP1:
	UF : 0, UT : 1,		CONFIG : 'N U T, 0, 0, 0',
	X = 1212.025  mm,	Y = -81.473  mm,	Z = -230.292  mm,
	W = 0.000 deg,	P = 30.000 deg,	R = -160.000 deg
};
P[189]{
   GP1:
	UF : 0, UT : 1,		CONFIG : 'N U T, 0, 0, 0',
	X = 1210.636  mm,	Y = -80.069  mm,	Z = -229.977  mm,
	W = 0.000 deg,	P = 30.000 deg,	R = -160.000 deg
};
P[190]{
   GP1:
	UF : 0, UT : 1,		CONFIG : 'N U T, 0, 0, 0',
	X = 1209.247  mm,	Y = -78.664  mm,	Z = -229.663  mm,
	W = 0.000 deg,	P = 30.000 deg,	R = -161.844 deg
};
P[191]{
   GP1:
	UF : 0, UT : 1,		CONFIG : 'N U T, 0, 0, 0',
	X = 1207.858  mm,	Y = -77.260  mm,	Z = -229.349  mm,
	W = 0.000 deg,	P = 30.000 deg,	R = -165.936 deg
};
P[192]{
   GP1:
	UF : 0, UT : 1,		CONFIG : 'N U T, 0, 0, 0',
	X = 1206.469  mm,	Y = -75.856  mm,	Z = -229.035  mm,
	W = 0.000 deg,	P = 30.000 deg,	R = -170.027 deg
};
P[193]{
   GP1:
	UF : 0, UT : 1,		CONFIG : 'N U T, 0, 0, 0',
	X = 1205.080  mm,	Y = -74.451  mm,	Z = -228.721  mm,
	W = 0.000 deg,	P = 30.000 deg,	R = -174.119 deg
};
P[194]{
   GP1:
	UF : 0, UT : 1,		CONFIG : 'N U T, 0, 0, 0',
	X = 1203.691  mm,	Y = -73.047  mm,	Z = -228.407  mm,
	W = 0.000 deg,	P = 30.000 deg,	R = -178.211 deg
};
P[195]{
   GP1:
	UF : 0, UT : 1,		CONFIG : 'N U T, 0, 0, 0',
	X = 1202.302  mm,	Y = -71.643  mm,	Z = -228.092  mm,
	W = 0.000 deg,	P = 30.000 deg,	R = 179.542 deg
};
P[196]{
   GP1:
	UF : 0, UT : 1,		CONFIG : 'N U T, 0, 0, 0',
	X = 1201.581  mm,	Y = -70.915  mm,	Z = -227.929  mm,
	W = 0.000 deg,	P = 30.000 deg,	R = 179.542 deg
};
P[197]{
   GP1:
	UF : 0, UT : 1,		CONFIG : 'N U T, 0, 0, 0',
	X = 1201.589  mm,	Y = -69.952  mm,	Z = -227.917  mm,
	W = 0.000 deg,	P = 30.000 deg,	R = 179.542 deg
};
P[198]{
   GP1:
	UF : 0, UT : 1,		CONFIG : 'N U T, 0, 0, 0',
	X = 1201.605  mm,	Y = -67.952  mm,	Z = -227.890  mm,
	W = 0.000 deg,	P = 30.000 deg,	R = 179.542 deg
};
P[199]{
   GP1:
	UF : 0, UT : 1,		CONFIG : 'N U T, 0, 0, 0',
	X = 1201.621  mm,	Y = -65.952  mm,	Z = -227.864  mm,
	W = 0.000 deg,	P = 30.000 deg,	R = 179.542 deg
};
P[200]{
   GP1:
	UF : 0, UT : 1,		CONFIG : 'N U T, 0, 0, 0',
	X = 1201.637  mm,	Y = -63.953  mm,	Z = -227.838  mm,
	W = 0.000 deg,	P = 30.000 deg,	R = 179.542 deg
};
P[201]{
   GP1:
	UF : 0, UT : 1,		CONFIG : 'N U T, 0, 0, 0',
	X = 1201.653  mm,	Y = -61.953  mm,	Z = -227.812  mm,
	W = 0.000 deg,	P = 30.000 deg,	R = 179.542 deg
};
P[202]{
   GP1:
	UF : 0, UT : 1,		CONFIG : 'N U T, 0, 0, 0',
	X = 1201.669  mm,	Y = -59.953  mm,	Z = -227.785  mm,
	W = 0.000 deg,	P = 30.000 deg,	R = 179.542 deg
};
P[203]{
   GP1:
	UF : 0, UT : 1,		CONFIG : 'N U T, 0, 0, 0',
	X = 1201.685  mm,	Y = -57.953  mm,	Z = -227.759  mm,
	W = 0.000 deg,	P = 30.000 deg,	R = 179.542 deg
};
P[204]{
   GP1:
	UF : 0, UT : 1,		CONFIG : 'N U T, 0, 0, 0',
	X = 1201.701  mm,	Y = -55.954  mm,	Z = -227.733  mm,
	W = 0.000 deg,	P = 30.000 deg,	R = 179.542 deg
};
P[205]{
   GP1:
	UF : 0, UT : 1,		CONFIG : 'N U T, 0, 0, 0',
	X = 1201.717  mm,	Y = -53.954  mm,	Z = -227.706  mm,
	W = 0.000 deg,	P = 30.000 deg,	R = 179.542 deg
};
P[206]{
   GP1:
	UF : 0, UT : 1,		CONFIG : 'N U T, 0, 0, 0',
	X = 1201.733  mm,	Y = -51.954  mm,	Z = -227.680  mm,
	W = 0.000 deg,	P = 30.000 deg,	R = 179.542 deg
};
P[207]{
   GP1:
	UF : 0, UT : 1,		CONFIG : 'N U T, 0, 0, 0',
	X = 1201.749  mm,	Y = -49.954  mm,	Z = -227.654  mm,
	W = 0.000 deg,	P = 30.000 deg,	R = 179.542 deg
};
P[208]{
   GP1:
	UF : 0, UT : 1,		CONFIG : 'N U T, 0, 0, 0',
	X = 1201.765  mm,	Y = -47.955  mm,	Z = -227.627  mm,
	W = 0.000 deg,	P = 30.000 deg,	R = 179.542 deg
};
P[209]{
   GP1:
	UF : 0, UT : 1,		CONFIG : 'N U T, 0, 0, 0',
	X = 1201.781  mm,	Y = -45.955  mm,	Z = -227.601  mm,
	W = 0.000 deg,	P = 30.000 deg,	R = 179.542 deg
};
P[210]{
   GP1:
	UF : 0, UT : 1,		CONFIG : 'N U T, 0, 0, 0',
	X = 1201.797  mm,	Y = -43.955  mm,	Z = -227.575  mm,
	W = 0.000 deg,	P = 30.000 deg,	R = 179.542 deg
};
P[211]{
   GP1:
	UF : 0, UT : 1,		CONFIG : 'N U T, 0, 0, 0',
	X = 1201.813  mm,	Y = -41.955  mm,	Z = -227.549  mm,
	W = 0.000 deg,	P = 30.000 deg,	R = 179.542 deg
};
P[212]{
   GP1:
	UF : 0, UT : 1,		CONFIG : 'N U T, 0, 0, 0',
	X = 1201.829  mm,	Y = -39.956  mm,	Z = -227.522  mm,
	W = 0.000 deg,	P = 30.000 deg,	R = 179.542 deg
};
P[213]{
   GP1:
	UF : 0, UT : 1,		CONFIG : 'N U T, 0, 0, 0',
	X = 1201.845  mm,	Y = -37.956  mm,	Z = -227.496  mm,
	W = 0.000 deg,	P = 30.000 deg,	R = 179.542 deg
};
P[214]{
   GP1:
	UF : 0, UT : 1,		CONFIG : 'N U T, 0, 0, 0',
	X = 1201.861  mm,	Y = -35.956  mm,	Z = -227.470  mm,
	W = 0.000 deg,	P = 30.000 deg,	R = 179.542 deg
};
P[215]{
   GP1:
	UF : 0, UT : 1,		CONFIG : 'N U T, 0, 0, 0',
	X = 1201.877  mm,	Y = -33.956  mm,	Z = -227.443  mm,
	W = 0.000 deg,	P = 30.000 deg,	R = 179.542 deg
};
P[216]{
   GP1:
	UF : 0, UT : 1,		CONFIG : 'N U T, 0, 0, 0',
	X = 1201.893  mm,	Y = -31.956  mm,	Z = -227.417  mm,
	W = 0.000 deg,	P = 30.000 deg,	R = 179.542 deg
};
P[217]{
   GP1:
	UF : 0, UT : 1,		CONFIG : 'N U T, 0, 0, 0',
	X = 1201.909  mm,	Y = -29.957  mm,	Z = -227.391  mm,
	W = 0.000 deg,	P = 30.000 deg,	R = 179.542 deg
};
P[218]{
   GP1:
	UF : 0, UT : 1,		CONFIG : 'N U T, 0, 0, 0',
	X = 1201.925  mm,	Y = -27.957  mm,	Z = -227.365  mm,
	W = 0.000 deg,	P = 30.000 deg,	R = 179.542 deg
};
P[219]{
   GP1:
	UF : 0, UT : 1,		CONFIG : 'N U T, 0, 0, 0',
	X = 1201.941  mm,	Y = -25.957  mm,	Z = -227.338  mm,
	W = 0.000 deg,	P = 30.000 deg,	R = 179.542 deg
};
P[220]{
   GP1:
	UF : 0, UT : 1,		CONFIG : 'N U T, 0, 0, 0',
	X = 1201.956  mm,	Y = -23.957  mm,	Z = -227.312  mm,
	W = 0.000 deg,	P = 30.000 deg,	R = 179.542 deg
};
P[221]{
   GP1:
	UF : 0, UT : 1,		CONFIG : 'N U T, 0, 0, 0',
	X = 1201.972  mm,	Y = -21.958  mm,	Z = -227.286  mm,
	W = 0.000 deg,	P = 30.000 deg,	R = 177.661 deg
};
P[222]{
   GP1:
	UF : 0, UT : 1,		CONFIG : 'N U T, 0, 0, 0',
	X = 1201.988  mm,	Y = -19.958  mm,	Z = -227.259  mm,
	W = 0.000 deg,	P = 30.000 deg,	R = 173.753 deg
};
P[223]{
   GP1:
	UF : 0, UT : 1,		CONFIG : 'N U T, 0, 0, 0',
	X = 1202.004  mm,	Y = -17.958  mm,	Z = -227.233  mm,
	W = 0.000 deg,	P = 30.000 deg,	R = 169.844 deg
};
P[224]{
   GP1:
	UF : 0, UT : 1,		CONFIG : 'N U T, 0, 0, 0',
	X = 1202.020  mm,	Y = -15.958  mm,	Z = -227.207  mm,
	W = 0.000 deg,	P = 30.000 deg,	R = 165.936 deg
};
P[225]{
   GP1:
	UF : 0, UT : 1,		CONFIG : 'N U T, 0, 0, 0',
	X = 1202.036  mm,	Y = -13.959  mm,	Z = -227.180  mm,
	W = 0.000 deg,	P = 30.000 deg,	R = 162.027 deg
};
P[226]{
   GP1:
	UF : 0, UT : 1,		CONFIG : 'N U T, 0, 0, 0',
	X = 1202.047  mm,	Y = -12.644  mm,	Z = -227.163  mm,
	W = 0.000 deg,	P = 30.000 deg,	R = 160.000 deg
};
P[227]{
   GP1:
	UF : 0, UT : 1,		CONFIG : 'N U T, 0, 0, 0',
	X = 1202.506  mm,	Y = -12.146  mm,	Z = -227.267  mm,
	W = 0.000 deg,	P = 30.000 deg,	R = 160.000 deg
};
P[228]{
   GP1:
	UF : 0, UT : 1,		CONFIG : 'N U T, 0, 0, 0',
	X = 1203.844  mm,	Y = -10.691  mm,	Z = -227.571  mm,
	W = 0.000 deg,	P = 30.000 deg,	R = 160.000 deg
};
P[229]{
   GP1:
	UF : 0, UT : 1,		CONFIG : 'N U T, 0, 0, 0',
	X = 1205.183  mm,	Y = -9.237  mm,	Z = -227.876  mm,
	W = 0.000 deg,	P = 30.000 deg,	R = 160.000 deg
};
P[230]{
   GP1:
	UF : 0, UT : 1,		CONFIG : 'N U T, 0, 0, 0',
	X = 1206.522  mm,	Y = -7.783  mm,	Z = -228.180  mm,
	W = 0.000 deg,	P = 30.000 deg,	R = 160.000 deg
};
P[231]{
   GP1:
	UF : 0, UT : 1,		CONFIG : 'N U T, 0, 0, 0',
	X = 1207.861  mm,	Y = -6.329  mm,	Z = -228.484  mm,
	W = 0.000 deg,	P = 30.000 deg,	R = 160.000 deg
};
P[232]{
   GP1:
	UF : 0, UT : 1,		CONFIG : 'N U T, 0, 0, 0',
	X = 1209.200  mm,	Y = -4.874  mm,	Z = -228.788  mm,
	W = 0.000 deg,	P = 30.000 deg,	R = 160.000 deg
};
P[233]{
   GP1:
	UF : 0, UT : 1,		CONFIG : 'N U T, 0, 0, 0',
	X = 1210.539  mm,	Y = -3.420  mm,	Z = -229.092  mm,
	W = 0.000 deg,	P = 30.000 deg,	R = 160.000 deg
};
P[234]{
   GP1:
	UF : 0, UT : 1,		CONFIG : 'N U T, 0, 0, 0',
	X = 1211.878  mm,	Y = -1.966  mm,	Z = -229.396  mm,
	W = 0.000 deg,	P = 30.000 deg,	R = 160.000 deg
};
P[235]{
   GP1:
	UF : 0, UT : 1,		CONFIG : 'N U T, 0, 0, 0',
	X = 1213.217  mm,	Y = -0.511  mm,	Z = -229.700  mm,
	W = 0.000 deg,	P = 30.000 deg,	R = 160.000 deg
};
P[236]{
   GP1:
	UF : 0, UT : 1,		CONFIG : 'N U T, 0, 0, 0',
	X = 1214.555  mm,	Y = 0.943  mm,	Z = -230.004  mm,
	W = 0.000 deg,	P = 30.000 deg,	R = 160.000 deg
};
P[237]{
   GP1:
	UF : 0, UT : 1,		CONFIG : 'N U T, 0, 0, 0',
	X = 1215.894  mm,	Y = 2.397  mm,	Z = -230.308  mm,
	W = 0.000 deg,	P = 30.000 deg,	R = 160.000 deg
};
P[238]{
   GP1:
	UF : 0, UT : 1,		CONFIG : 'N U T, 0, 0, 0',
	X = 1217.233  mm,	Y = 3.851  mm,	Z = -230.612  mm,
	W = 0.000 deg,	P = 30.000 deg,	R = 160.000 deg
};
P[239]{
   GP1:
	UF : 0, UT : 1,		CONFIG : 'N U T, 0, 0, 0',
	X = 1218.572  mm,	Y = 5.306  mm,	Z = -230.916  mm,
	W = 0.000 deg,	P = 30.000 deg,	R = 160.000 deg
};
P[240]{
   GP1:
	UF : 0, UT : 1,		CONFIG : 'N U T, 0, 0, 0',
	X = 1219.911  mm,	Y = 6.760  mm,	Z = -231.220  mm,
	W = 0.000 deg,	P = 30.000 deg,	R = 160.000 deg
};
P[241]{
   GP1:
	UF : 0, UT : 1,		CONFIG : 'N U T, 0, 0, 0',
	X = 1221.250  mm,	Y = 8.214  mm,	Z = -231.524  mm,
	W = 0.000 deg,	P = 30.000 deg,	R = 160.000 deg
};
P[242]{
   GP1:
	UF : 0, UT : 1,		CONFIG : 'N U T, 0, 0, 0',
	X = 1222.589  mm,	Y = 9.668  mm,	Z = -231.829  mm,
	W = 0.000 deg,	P = 30.000 deg,	R = 160.000 deg
};
P[243]{
   GP1:
	UF : 0, UT : 1,		CONFIG : 'N U T, 0, 0, 0',
	X = 1223.928  mm,	Y = 11.123  mm,	Z = -232.133  mm,
	W = 0.000 deg,	P = 30.000 deg,	R = 160.000 deg
};
P[244]{
   GP1:
	UF : 0, UT : 1,		CONFIG : 'N U T, 0, 0, 0',
	X = 1225.267  mm,	Y = 12.577  mm,	Z = -232.437  mm,
	W = 0.000 deg,	P = 30.000 deg,	R = 160.000 deg
};
P[245]{
   GP1:
	UF : 0, UT : 1,		CONFIG : 'N U T, 0, 0, 0',
	X = 1226.605  mm,	Y = 14.031  mm,	Z = -232.741  mm,
	W = 0.000 deg,	P = 30.000 deg,	R = 160.000 deg
};
P[246]{
   GP1:
	UF : 0, UT : 1,		CONFIG : 'N U T, 0, 0, 0',
	X = 1227.944  mm,	Y = 15.486  mm,	Z = -233.045  mm,
	W = 0.000 deg,	P = 30.000 deg,	R = 160.000 deg
};
P[247]{
   GP1:
	UF : 0, UT : 1,		CONFIG : 'N U T, 0, 0, 0',
	X = 1229.283  mm,	Y = 16.940  mm,	Z = -233.349  mm,
	W = 0.000 deg,	P = 30.000 deg,	R = 160.000 deg
};
P[248]{
   GP1:
	UF : 0, UT : 1,		CONFIG : 'N U T, 0, 0, 0',
	X = 1230.622  mm,	Y = 18.394  mm,	Z = -233.653  mm,
	W = 0.000 deg,	P = 30.000 deg,	R = 165.983 deg
};
P[249]{
   GP1:
	UF : 0, UT : 1,		CONFIG : 'N U T, 0, 0, 0',
	X = 1231.961  mm,	Y = 19.848  mm,	Z = -233.957  mm,
	W = 0.000 deg,	P = 30.000 deg,	R = 170.439 deg
};
P[250]{
   GP1:
	UF : 0, UT : 1,		CONFIG : 'N U T, 0, 0, 0',
	X = 1233.300  mm,	Y = 21.303  mm,	Z = -234.261  mm,
	W = 0.000 deg,	P = 30.000 deg,	R = 174.895 deg
};
P[251]{
   GP1:
	UF : 0, UT : 1,		CONFIG : 'N U T, 0, 0, 0',
	X = 1234.639  mm,	Y = 22.757  mm,	Z = -234.565  mm,
	W = 0.000 deg,	P = 30.000 deg,	R = 179.351 deg
};
P[252]{
   GP1:
	UF : 0, UT : 1,		CONFIG : 'N U T, 0, 0, 0',
	X = 1235.978  mm,	Y = 24.211  mm,	Z = -234.869  mm,
	W = 0.000 deg,	P = 30.000 deg,	R = -177.720 deg
};
P[253]{
   GP1:
	UF : 0, UT : 1,		CONFIG : 'N U T, 0, 0, 0',
	X = 1236.091  mm,	Y = 24.335  mm,	Z = -234.895  mm,
	W = 0.000 deg,	P = 30.000 deg,	R = -177.720 deg
};
P[254]{
   GP1:
	UF : 0, UT : 1,		CONFIG : 'N U T, 0, 0, 0',
	X = 1236.019  mm,	Y = 26.163  mm,	Z = -234.864  mm,
	W = 0.000 deg,	P = 30.000 deg,	R = -177.720 deg
};
P[255]{
   GP1:
	UF : 0, UT : 1,		CONFIG : 'N U T, 0, 0, 0',
	X = 1235.939  mm,	Y = 28.161  mm,	Z = -234.829  mm,
	W = 0.000 deg,	P = 30.000 deg,	R = -177.720 deg
};
P[256]{
   GP1:
	UF : 0, UT : 1,		CONFIG : 'N U T, 0, 0, 0',
	X = 1235.860  mm,	Y = 30.159  mm,	Z = -234.794  mm,
	W = 0.000 deg,	P = 30.000 deg,	R = -177.720 deg
};
P[257]{
   GP1:
	UF : 0, UT : 1,		CONFIG : 'N U T, 0, 0, 0',
	X = 1235.780  mm,	Y = 32.157  mm,	Z = -234.760  mm,
	W = 0.000 deg,	P = 30.000 deg,	R = -177.720 deg
};
P[258]{
   GP1:
	UF : 0, UT : 1,		CONFIG : 'N U T, 0, 0, 0',
	X = 1235.700  mm,	Y = 34.156  mm,	Z = -234.725  mm,
	W = 0.000 deg,	P = 30.000 deg,	R = -177.720 deg
};
P[259]{
   GP1:
	UF : 0, UT : 1,		CONFIG : 'N U T, 0, 0, 0',
	X = 1235.621  mm,	Y = 36.154  mm,	Z = -234.691  mm,
	W = 0.000 deg,	P = 30.000 deg,	R = -177.720 deg
};
P[260]{
   GP1:
	UF : 0, UT : 1,		CONFIG : 'N U T, 0, 0, 0',
	X = 1235.541  mm,	Y = 38.152  mm,	Z = -234.656  mm,
	W = 0.000 deg,	P = 30.000 deg,	R = -177.720 deg
};
P[261]{
   GP1:
	UF : 0, UT : 1,		CONFIG : 'N U T, 0, 0, 0',
	X = 1235.462  mm,	Y = 40.150  mm,	Z = -234.622  mm,
	W = 0.000 deg,	P = 30.000 deg,	R = -177.720 deg
};
P[262]{
   GP1:
	UF : 0, UT : 1,		CONFIG : 'N U T, 0, 0, 0',
	X = 1235.382  mm,	Y = 42.148  mm,	Z = -234.587  mm,
	W = 0.000 deg,	P = 30.000 deg,	R = -177.720 deg
};
P[263]{
   GP1:
	UF : 0, UT : 1,		CONFIG : 'N U T, 0, 0, 0',
	X = 1235.303  mm,	Y = 44.146  mm,	Z = -234.552  mm,
	W = 0.000 deg,	P = 30.000 deg,	R = -177.720 deg
};
P[264]{
   GP1:
	UF : 0, UT : 1,		CONFIG : 'N U T, 0, 0, 0',
	X = 1235.223  mm,	Y = 46.144  mm,	Z = -234.518  mm,
	W = 0.000 deg,	P = 30.000 deg,	R = -177.720 deg
};
P[265]{
   GP1:
	UF : 0, UT : 1,		CONFIG : 'N U T, 0, 0, 0',
	X = 1235.143  mm,	Y = 48.142  mm,	Z = -234.483  mm,
	W = 0.000 deg,	P = 30.000 deg,	R = -177.720 deg
};
P[266]{
   GP1:
	UF : 0, UT : 1,		CONFIG : 'N U T, 0, 0, 0',
	X = 1235.064  mm,	Y = 50.141  mm,	Z = -234.449  mm,
	W = 0.000 deg,	P = 30.000 deg,	R = -177.720 deg
};
P[267]{
   GP1:
	UF : 0, UT : 1,		CONFIG : 'N U T, 0, 0, 0',
	X = 1234.984  mm,	Y = 52.139  mm,	Z = -234.414  mm,
	W = 0.000 deg,	P = 30.000 deg,	R = -177.720 deg
};
P[268]{
   GP1:
	UF : 0, UT : 1,		CONFIG : 'N U T, 0, 0, 0',
	X = 1234.905  mm,	Y = 54.137  mm,	Z = -234.380  mm,
	W = 0.000 deg,	P = 30.000 deg,	R = -177.720 deg
};
P[269]{
   GP1:
	UF : 0, UT : 1,		CONFIG : 'N U T, 0, 0, 0',
	X = 1234.825  mm,	Y = 56.135  mm,	Z = -234.345  mm,
	W = 0.000 deg,	P = 30.000 deg,	R = -177.720 deg
};
P[270]{
   GP1:
	UF : 0, UT : 1,		CONFIG : 'N U T, 0, 0, 0',
	X = 1234.746  mm,	Y = 58.133  mm,	Z = -234.310  mm,
	W = 0.000 deg,	P = 30.000 deg,	R = -177.720 deg
};
P[271]{
   GP1:
	UF : 0, UT : 1,		CONFIG : 'N U T, 0, 0, 0',
	X = 1234.666  mm,	Y = 60.131  mm,	Z = -234.276  mm,
	W = 0.000 deg,	P = 30.000 deg,	R = -177.720 deg
};
P[272]{
   GP1:
	UF : 0, UT : 1,		CONFIG : 'N U T, 0, 0, 0',
	X = 1234.586  mm,	Y = 62.129  mm,	Z = -234.241  mm,
	W = 0.000 deg,	P = 30.000 deg,	R = -177.720 deg
};
P[273]{
   GP1:
	UF : 0, UT : 1,		CONFIG : 'N U T, 0, 0, 0',
	X = 1234.507  mm,	Y = 64.127  mm,	Z = -234.207  mm,
	W = 0.000 deg,	P = 30.000 deg,	R = -177.720 deg
};
P[274]{
   GP1:
	UF : 0, UT : 1,		CONFIG : 'N U T, 0, 0, 0',
	X = 1234.427  mm,	Y = 66.125  mm,	Z = -234.172  mm,
	W = 0.000 deg,	P = 30.000 deg,	R = -177.720 deg
};
P[275]{
   GP1:
	UF : 0, UT : 1,		CONFIG : 'N U T, 0, 0, 0',
	X = 1234.348  mm,	Y = 68.124  mm,	Z = -234.138  mm,
	W = 0.000 deg,	P = 30.000 deg,	R = -177.720 deg
};
P[276]{
   GP1:
	UF : 0, UT : 1,		CONFIG : 'N U T, 0, 0, 0',
	X = 1234.268  mm,	Y = 70.122  mm,	Z = -234.103  mm,
	W = 0.000 deg,	P = 30.000 deg,	R = -177.720 deg
};
P[277]{
   GP1:
	UF : 0, UT : 1,		CONFIG : 'N U T, 0, 0, 0',
	X = 1234.189  mm,	Y = 72.120  mm,	Z = -234.068  mm,
	W = 0.000 deg,	P = 30.000 deg,	R = -177.720 deg
};
P[278]{
   GP1:
	UF : 0, UT : 1,		CONFIG : 'N U T, 0, 0, 0',
	X = 1234.109  mm,	Y = 74.118  mm,	Z = -234.034  mm,
	W = 0.000 deg,	P = 30.000 deg,	R = -170.933 deg
};
P[279]{
   GP1:
	UF : 0, UT : 1,		CONFIG : 'N U T, 0, 0, 0',
	X = 1234.029  mm,	Y = 76.116  mm,	Z = -233.999  mm,
	W = 0.000 deg,	P = 30.000 deg,	R = -167.389 deg
};
P[280]{
   GP1:
	UF : 0, UT : 1,		CONFIG : 'N U T, 0, 0, 0',
	X = 1233.950  mm,	Y = 78.114  mm,	Z = -233.965  mm,
	W = 0.000 deg,	P = 30.000 deg,	R = -163.845 deg
};
P[281]{
   GP1:
	UF : 0, UT : 1,		CONFIG : 'N U T, 0, 0, 0',
	X = 1233.870  mm,	Y = 80.112  mm,	Z = -233.930  mm,
	W = 0.000 deg,	P = 30.000 deg,	R = -160.301 deg
};
P[282]{
   GP1:
	UF : 0, UT : 1,		CONFIG : 'N U T, 0, 0, 0',
	X = 1233.805  mm,	Y = 81.755  mm,	Z = -233.902  mm,
	W = 0.000 deg,	P = 30.000 deg,	R = -160.000 deg
};
P[283]{
   GP1:
	UF : 0, UT : 1,		CONFIG : 'N U T, 0, 0, 0',
	X = 1233.555  mm,	Y = 82.001  mm,	Z = -233.843  mm,
	W = 0.000 deg,	P = 30.000 deg,	R = -160.000 deg
};
P[284]{
   GP1:
	UF : 0, UT : 1,		CONFIG : 'N U T, 0, 0, 0',
	X = 1232.150  mm,	Y = 83.385  mm,	Z = -233.510  mm,
	W = 0.000 deg,	P = 30.000 deg,	R = -160.000 deg
};
P[285]{
   GP1:
	UF : 0, UT : 1,		CONFIG : 'N U T, 0, 0, 0',
	X = 1230.746  mm,	Y = 84.770  mm,	Z = -233.177  mm,
	W = 0.000 deg,	P = 30.000 deg,	R = -160.000 deg
};
P[286]{
   GP1:
	UF : 0, UT : 1,		CONFIG : 'N U T, 0, 0, 0',
	X = 1229.341  mm,	Y = 86.154  mm,	Z = -232.845  mm,
	W = 0.000 deg,	P = 30.000 deg,	R = -160.000 deg
};
P[287]{
   GP1:
	UF : 0, UT : 1,		CONFIG : 'N U T, 0, 0, 0',
	X = 1227.936  mm,	Y = 87.538  mm,	Z = -232.512  mm,
	W = 0.000 deg,	P = 30.000 deg,	R = -160.000 deg
};
P[288]{
   GP1:
	UF : 0, UT : 1,		CONFIG : 'N U T, 0, 0, 0',
	X = 1226.531  mm,	Y = 88.922  mm,	Z = -232.180  mm,
	W = 0.000 deg,	P = 30.000 deg,	R = -160.000 deg
};
P[289]{
   GP1:
	UF : 0, UT : 1,		CONFIG : 'N U T, 0, 0, 0',
	X = 1225.126  mm,	Y = 90.306  mm,	Z = -231.847  mm,
	W = 0.000 deg,	P = 30.000 deg,	R = -160.000 deg
};
P[290]{
   GP1:
	UF : 0, UT : 1,		CONFIG : 'N U T, 0, 0, 0',
	X = 1223.722  mm,	Y = 91.690  mm,	Z = -231.514  mm,
	W = 0.000 deg,	P = 30.000 deg,	R = -160.000 deg
};
P[291]{
   GP1:
	UF : 0, UT : 1,		CONFIG : 'N U T, 0, 0, 0',
	X = 1222.317  mm,	Y = 93.075  mm,	Z = -231.182  mm,
	W = 0.000 deg,	P = 30.000 deg,	R = -160.000 deg
};
P[292]{
   GP1:
	UF : 0, UT : 1,		CONFIG : 'N U T, 0, 0, 0',
	X = 1220.912  mm,	Y = 94.459  mm,	Z = -230.849  mm,
	W = 0.000 deg,	P = 30.000 deg,	R = -160.000 deg
};
P[293]{
   GP1:
	UF : 0, UT : 1,		CONFIG : 'N U T, 0, 0, 0',
	X = 1219.507  mm,	Y = 95.843  mm,	Z = -230.517  mm,
	W = 0.000 deg,	P = 30.000 deg,	R = -160.000 deg
};
P[294]{
   GP1:
	UF : 0, UT : 1,		CONFIG : 'N U T, 0, 0, 0',
	X = 1218.102  mm,	Y = 97.227  mm,	Z = -230.184  mm,
	W = 0.000 deg,	P = 30.000 deg,	R = -160.000 deg
};
P[295]{
   GP1:
	UF : 0, UT : 1,		CONFIG : 'N U T, 0, 0, 0',
	X = 1216.697  mm,	Y = 98.611  mm,	Z = -229.851  mm,
	W = 0.000 deg,	P = 30.000 deg,	R = -160.000 deg
};
P[296]{
   GP1:
	UF : 0, UT : 1,		CONFIG : 'N U T, 0, 0, 0',
	X = 1215.293  mm,	Y = 99.995  mm,	Z = -229.519  mm,
	W = 0.000 deg,	P = 30.000 deg,	R = -160.000 deg
};
P[297]{
   GP1:
	UF : 0, UT : 1,		CONFIG : 'N U T, 0, 0, 0',
	X = 1213.888  mm,	Y = 101.379  mm,	Z = -229.186  mm,
	W = 0.000 deg,	P = 30.000 deg,	R = -160.000 deg
};
P[298]{
   GP1:
	UF : 0, UT : 1,		CONFIG : 'N U T, 0, 0, 0',
	X = 1212.483  mm,	Y = 102.764  mm,	Z = -228.854  mm,
	W = 0.000 deg,	P = 30.000 deg,	R = -160.000 deg
};
P[299]{
   GP1:
	UF : 0, UT : 1,		CONFIG : 'N U T, 0, 0, 0',
	X = 1211.078  mm,	Y = 104.148  mm,	Z = -228.521  mm,
	W = 0.000 deg,	P = 30.000 deg,	R = -160.000 deg
};
P[300]{
   GP1:
	UF : 0, UT : 1,		CONFIG : 'N U T, 0, 0, 0',
	X = 1209.673  mm,	Y = 105.532  mm,	Z = -228.188  mm,
	W = 0.000 deg,	P = 30.000 deg,	R = -160.000 deg
};
P[301]{
   GP1:
	UF : 0, UT : 1,		CONFIG : 'N U T, 0, 0, 0',
	X = 1208.269  mm,	Y = 106.916  mm,	Z = -227.856  mm,
	W = 0.000 deg,	P = 30.000 deg,	R = -160.000 deg
};
P[302]{
   GP1:
	UF : 0, UT : 1,		CONFIG : 'N U T, 0, 0, 0',
	X = 1206.864  mm,	Y = 108.300  mm,	Z = -227.523  mm,
	W = 0.000 deg,	P = 30.000 deg,	R = -160.000 deg
};
P[303]{
   GP1:
	UF : 0, UT : 1,		CONFIG : 'N U T, 0, 0, 0',
	X = 1205.459  mm,	Y = 109.684  mm,	Z = -227.191  mm,
	W = 0.000 deg,	P = 30.000 deg,	R = -160.710 deg
};
P[304]{
   GP1:
	UF : 0, UT : 1,		CONFIG : 'N U T, 0, 0, 0',
	X = 1204.054  mm,	Y = 111.069  mm,	Z = -226.858  mm,
	W = 0.000 deg,	P = 30.000 deg,	R = -164.708 deg
};
P[305]{
   GP1:
	UF : 0, UT : 1,		CONFIG : 'N U T, 0, 0, 0',
	X = 1202.649  mm,	Y = 112.453  mm,	Z = -226.526  mm,
	W = 0.000 deg,	P = 30.000 deg,	R = -168.705 deg
};
P[306]{
   GP1:
	UF : 0, UT : 1,		CONFIG : 'N U T, 0, 0, 0',
	X = 1201.245  mm,	Y = 113.837  mm,	Z = -226.193  mm,
	W = 0.000 deg,	P = 30.000 deg,	R = -172.703 deg
};
P[307]{
   GP1:
	UF : 0, UT : 1,		CONFIG : 'N U T, 0, 0, 0',
	X = 1199.840  mm,	Y = 115.221  mm,	Z = -225.860  mm,
	W = 0.000 deg,	P = 30.000 deg,	R = -176.700 deg
};
P[308]{
   GP1:
	UF : 0, UT : 1,		CONFIG : 'N U T, 0, 0, 0',
	X = 1198.476  mm,	Y = 116.565  mm,	Z = -225.537  mm,
	W = 0.000 deg,	P = 30.000 deg,	R = -179.988 deg
};
P[309]{
   GP1:
	UF : 0, UT : 1,		CONFIG : 'N U T, 0, 0, 0',
	X = 1198.476  mm,	Y = 116.623  mm,	Z = -225.537  mm,
	W = 0.000 deg,	P = 30.000 deg,	R = -179.988 deg
};
P[310]{
   GP1:
	UF : 0, UT : 1,		CONFIG : 'N U T, 0, 0, 0',
	X = 1198.476  mm,	Y = 118.623  mm,	Z = -225.516  mm,
	W = 0.000 deg,	P = 30.000 deg,	R = -179.988 deg
};
P[311]{
   GP1:
	UF : 0, UT : 1,		CONFIG : 'N U T, 0, 0, 0',
	X = 1198.475  mm,	Y = 120.623  mm,	Z = -225.495  mm,
	W = 0.000 deg,	P = 30.000 deg,	R = -179.988 deg
};
P[312]{
   GP1:
	UF : 0, UT : 1,		CONFIG : 'N U T, 0, 0, 0',
	X = 1198.475  mm,	Y = 122.623  mm,	Z = -225.473  mm,
	W = 0.000 deg,	P = 30.000 deg,	R = -179.988 deg
};
P[313]{
   GP1:
	UF : 0, UT : 1,		CONFIG : 'N U T, 0, 0, 0',
	X = 1198.474  mm,	Y = 124.623  mm,	Z = -225.452  mm,
	W = 0.000 deg,	P = 30.000 deg,	R = -179.988 deg
};
P[314]{
   GP1:
	UF : 0, UT : 1,		CONFIG : 'N U T, 0, 0, 0',
	X = 1198.474  mm,	Y = 126.623  mm,	Z = -225.431  mm,
	W = 0.000 deg,	P = 30.000 deg,	R = -179.988 deg
};
P[315]{
   GP1:
	UF : 0, UT : 1,		CONFIG : 'N U T, 0, 0, 0',
	X = 1198.473  mm,	Y = 128.622  mm,	Z = -225.410  mm,
	W = 0.000 deg,	P = 30.000 deg,	R = -179.988 deg
};
P[316]{
   GP1:
	UF : 0, UT : 1,		CONFIG : 'N U T, 0, 0, 0',
	X = 1198.473  mm,	Y = 130.622  mm,	Z = -225.389  mm,
	W = 0.000 deg,	P = 30.000 deg,	R = -179.988 deg
};
P[317]{
   GP1:
	UF : 0, UT : 1,		CONFIG : 'N U T, 0, 0, 0',
	X = 1198.473  mm,	Y = 132.622  mm,	Z = -225.368  mm,
	W = 0.000 deg,	P = 30.000 deg,	R = -179.988 deg
};
P[318]{
   GP1:
	UF : 0, UT : 1,		CONFIG : 'N U T, 0, 0, 0',
	X = 1198.472  mm,	Y = 134.622  mm,	Z = -225.347  mm,
	W = 0.000 deg,	P = 30.000 deg,	R = -179.988 deg
};
P[319]{
   GP1:
	UF : 0, UT : 1,		CONFIG : 'N U T, 0, 0, 0',
	X = 1198.472  mm,	Y = 136.622  mm,	Z = -225.325  mm,
	W = 0.000 deg,	P = 30.000 deg,	R = -179.988 deg
};
P[320]{
   GP1:
	UF : 0, UT : 1,		CONFIG : 'N U T, 0, 0, 0',
	X = 1198.471  mm,	Y = 138.622  mm,	Z = -225.304  mm,
	W = 0.000 deg,	P = 30.000 deg,	R = -179.988 deg
};
P[321]{
   GP1:
	UF : 0, UT : 1,		CONFIG : 'N U T, 0, 0, 0',
	X = 1198.471  mm,	Y = 140.622  mm,	Z = -225.283  mm,
	W = 0.000 deg,	P = 30.000 deg,	R = -179.988 deg
};
P[322]{
   GP1:
	UF : 0, UT : 1,		CONFIG : 'N U T, 0, 0, 0',
	X = 1198.470  mm,	Y = 142.622  mm,	Z = -225.262  mm,
	W = 0.000 deg,	P = 30.000 deg,	R = -179.988 deg
};
P[323]{
   GP1:
	UF : 0, UT : 1,		CONFIG : 'N U T, 0, 0, 0',
	X = 1198.470  mm,	Y = 144.622  mm,	Z = -225.241  mm,
	W = 0.000 deg,	P = 30.000 deg,	R = -179.988 deg
};
P[324]{
   GP1:
	UF : 0, UT : 1,		CONFIG : 'N U T, 0, 0, 0',
	X = 1198.469  mm,	Y = 146.621  mm,	Z = -225.220  mm,
	W = 0.000 deg,	P = 30.000 deg,	R = -179.988 deg
};
P[325]{
   GP1:
	UF : 0, UT : 1,		CONFIG : 'N U T, 0, 0, 0',
	X = 1198.469  mm,	Y = 148.621  mm,	Z = -225.199  mm,
	W = 0.000 deg,	P = 30.000 deg,	R = -179.988 deg
};
P[326]{
   GP1:
	UF : 0, UT : 1,		CONFIG : 'N U T, 0, 0, 0',
	X = 1198.469  mm,	Y = 150.621  mm,	Z = -225.177  mm,
	W = 0.000 deg,	P = 30.000 deg,	R = -179.988 deg
};
P[327]{
   GP1:
	UF : 0, UT : 1,		CONFIG : 'N U T, 0, 0, 0',
	X = 1198.468  mm,	Y = 152.621  mm,	Z = -225.156  mm,
	W = 0.000 deg,	P = 30.000 deg,	R = -179.988 deg
};
P[328]{
   GP1:
	UF : 0, UT : 1,		CONFIG : 'N U T, 0, 0, 0',
	X = 1198.468  mm,	Y = 154.621  mm,	Z = -225.135  mm,
	W = 0.000 deg,	P = 30.000 deg,	R = -179.988 deg
};
P[329]{
   GP1:
	UF : 0, UT : 1,		CONFIG : 'N U T, 0, 0, 0',
	X = 1198.467  mm,	Y = 156.621  mm,	Z = -225.114  mm,
	W = 0.000 deg,	P = 30.000 deg,	R = -179.988 deg
};
P[330]{
   GP1:
	UF : 0, UT : 1,		CONFIG : 'N U T, 0, 0, 0',
	X = 1198.467  mm,	Y = 158.621  mm,	Z = -225.093  mm,
	W = 0.000 deg,	P = 30.000 deg,	R = -179.988 deg
};
P[331]{
   GP1:
	UF : 0, UT : 1,		CONFIG : 'N U T, 0, 0, 0',
	X = 1198.466  mm,	Y = 160.621  mm,	Z = -225.072  mm,
	W = 0.000 deg,	P = 30.000 deg,	R = -179.988 deg
};
P[332]{
   GP1:
	UF : 0, UT : 1,		CONFIG : 'N U T, 0, 0, 0',
	X = 1198.466  mm,	Y = 162.621  mm,	Z = -225.051  mm,
	W = 0.000 deg,	P = 30.000 deg,	R = -179.988 deg
};
P[333]{
   GP1:
	UF : 0, UT : 1,		CONFIG : 'N U T, 0, 0, 0',
	X = 1198.466  mm,	Y = 164.620  mm,	Z = -225.029  mm,
	W = 0.000 deg,	P = 30.000 deg,	R = -179.988 deg
};
P[334]{
   GP1:
	UF : 0, UT : 1,		CONFIG : 'N U T, 0, 0, 0',
	X = 1198.465  mm,	Y = 166.620  mm,	Z = -225.008  mm,
	W = 0.000 deg,	P = 30.000 deg,	R = -179.988 deg
};
P[335]{
   GP1:
	UF : 0, UT : 1,		CONFIG : 'N U T, 0, 0, 0',
	X = 1198.465  mm,	Y = 168.620  mm,	Z = -224.987  mm,
	W = 0.000 deg,	P = 30.000 deg,	R = 175.893 deg
};
P[336]{
   GP1:
	UF : 0, UT : 1,		CONFIG : 'N U T, 0, 0, 0',
	X = 1198.464  mm,	Y = 170.620  mm,	Z = -224.966  mm,
	W = 0.000 deg,	P = 30.000 deg,	R = 171.890 deg
};
P[337]{
   GP1:
	UF : 0, UT : 1,		CONFIG : 'N U T, 0, 0, 0',
	X = 1198.464  mm,	Y = 172.620  mm,	Z = -224.945  mm,
	W = 0.000 deg,	P = 30.000 deg,	R = 167.888 deg
};
P[338]{
   GP1:
	UF : 0, UT : 1,		CONFIG : 'N U T, 0, 0, 0',
	X = 1198.463  mm,	Y = 174.620  mm,	Z = -224.924  mm,
	W = 0.000 deg,	P = 30.000 deg,	R = 163.885 deg
};
P[339]{
   GP1:
	UF : 0, UT : 1,		CONFIG : 'N U T, 0, 0, 0',
	X = 1198.463  mm,	Y = 176.620  mm,	Z = -224.902  mm,
	W = 0.000 deg,	P = 30.000 deg,	R = 160.000 deg
};
P[340]{
   GP1:
	UF : 0, UT : 1,		CONFIG : 'N U T, 0, 0, 0',
	X = 1198.463  mm,	Y = 176.878  mm,	Z = -224.900  mm,
	W = 0.000 deg,	P = 30.000 deg,	R = 160.000 deg
};
P[341]{
   GP1:
	UF : 0, UT : 1,		CONFIG : 'N U T, 0, 0, 0',
	X = 1199.652  mm,	Y = 178.119  mm,	Z = -225.180  mm,
	W = 0.000 deg,	P = 30.000 deg,	R = 160.000 deg
};
P[342]{
   GP1:
	UF : 0, UT : 1,		CONFIG : 'N U T, 0, 0, 0',
	X = 1201.018  mm,	Y = 179.544  mm,	Z = -225.502  mm,
	W = 0.000 deg,	P = 30.000 deg,	R = 160.000 deg
};
P[343]{
   GP1:
	UF : 0, UT : 1,		CONFIG : 'N U T, 0, 0, 0',
	X = 1202.384  mm,	Y = 180.970  mm,	Z = -225.824  mm,
	W = 0.000 deg,	P = 30.000 deg,	R = 160.000 deg
};
P[344]{
   GP1:
	UF : 0, UT : 1,		CONFIG : 'N U T, 0, 0, 0',
	X = 1203.749  mm,	Y = 182.395  mm,	Z = -226.146  mm,
	W = 0.000 deg,	P = 30.000 deg,	R = 160.000 deg
};
P[345]{
   GP1:
	UF : 0, UT : 1,		CONFIG : 'N U T, 0, 0, 0',
	X = 1205.115  mm,	Y = 183.820  mm,	Z = -226.468  mm,
	W = 0.000 deg,	P = 30.000 deg,	R = 160.000 deg
};
P[346]{
   GP1:
	UF : 0, UT : 1,		CONFIG : 'N U T, 0, 0, 0',
	X = 1206.481  mm,	Y = 185.245  mm,	Z = -226.790  mm,
	W = 0.000 deg,	P = 30.000 deg,	R = 160.000 deg
};
P[347]{
   GP1:
	UF : 0, UT : 1,		CONFIG : 'N U T, 0, 0, 0',
	X = 1207.847  mm,	Y = 186.670  mm,	Z = -227.112  mm,
	W = 0.000 deg,	P = 30.000 deg,	R = 160.000 deg
};
P[348]{
   GP1:
	UF : 0, UT : 1,		CONFIG : 'N U T, 0, 0, 0',
	X = 1209.212  mm,	Y = 188.095  mm,	Z = -227.434  mm,
	W = 0.000 deg,	P = 30.000 deg,	R = 160.000 deg
};
P[349]{
   GP1:
	UF : 0, UT : 1,		CONFIG : 'N U T, 0, 0, 0',
	X = 1210.578  mm,	Y = 189.520  mm,	Z = -227.756  mm,
	W = 0.000 deg,	P = 30.000 deg,	R = 160.000 deg
};
P[350]{
   GP1:
	UF : 0, UT : 1,		CONFIG : 'N U T, 0, 0, 0',
	X = 1211.944  mm,	Y = 190.946  mm,	Z = -228.078  mm,
	W = 0.000 deg,	P = 30.000 deg,	R = 160.000 deg
};
P[351]{
   GP1:
	UF : 0, UT : 1,		CONFIG : 'N U T, 0, 0, 0',
	X = 1213.310  mm,	Y = 192.371  mm,	Z = -228.400  mm,
	W = 0.000 deg,	P = 30.000 deg,	R = 160.000 deg
};
P[352]{
   GP1:
	UF : 0, UT : 1,		CONFIG : 'N U T, 0, 0, 0',
	X = 1214.675  mm,	Y = 193.796  mm,	Z = -228.722  mm,
	W = 0.000 deg,	P = 30.000 deg,	R = 160.000 deg
};
P[353]{
   GP1:
	UF : 0, UT : 1,		CONFIG : 'N U T, 0, 0, 0',
	X = 1216.041  mm,	Y = 195.221  mm,	Z = -229.044  mm,
	W = 0.000 deg,	P = 30.000 deg,	R = 160.000 deg
};
P[354]{
   GP1:
	UF : 0, UT : 1,		CONFIG : 'N U T, 0, 0, 0',
	X = 1217.407  mm,	Y = 196.646  mm,	Z = -229.366  mm,
	W = 0.000 deg,	P = 30.000 deg,	R = 160.000 deg
};
P[355]{
   GP1:
	UF : 0, UT : 1,		CONFIG : 'N U T, 0, 0, 0',
	X = 1218.773  mm,	Y = 198.071  mm,	Z = -229.688  mm,
	W = 0.000 deg,	P = 30.000 deg,	R = 160.000 deg
};
P[356]{
   GP1:
	UF : 0, UT : 1,		CONFIG : 'N U T, 0, 0, 0',
	X = 1220.138  mm,	Y = 199.497  mm,	Z = -230.010  mm,
	W = 0.000 deg,	P = 30.000 deg,	R = 160.000 deg
};
P[357]{
   GP1:
	UF : 0, UT : 1,		CONFIG : 'N U T, 0, 0, 0',
	X = 1221.504  mm,	Y = 200.922  mm,	Z = -230.332  mm,
	W = 0.000 deg,	P = 30.000 deg,	R = 160.000 deg
};
P[358]{
   GP1:
	UF : 0, UT : 1,		CONFIG : 'N U T, 0, 0, 0',
	X = 1222.870  mm,	Y = 202.347  mm,	Z = -230.654  mm,
	W = 0.000 deg,	P = 30.000 deg,	R = 160.000 deg
};
P[359]{
   GP1:
	UF : 0, UT : 1,		CONFIG : 'N U T, 0, 0, 0',
	X = 1224.236  mm,	Y = 203.772  mm,	Z = -230.976  mm,
	W = 0.000 deg,	P = 30.000 deg,	R = 160.000 deg
};
P[360]{
   GP1:
	UF : 0, UT : 1,		CONFIG : 'N U T, 0, 0, 0',
	X = 1225.601  mm,	Y = 205.197  mm,	Z = -231.298  mm,
	W = 0.000 deg,	P = 30.000 deg,	R = 160.000 deg
};
P[361]{
   GP1:
	UF : 0, UT : 1,		CONFIG : 'N U T, 0, 0, 0',
	X = 1226.967  mm,	Y = 206.622  mm,	Z = -231.620  mm,
	W = 0.000 deg,	P = 30.000 deg,	R = 163.555 deg
};
P[362]{
   GP1:
	UF : 0, UT : 1,		CONFIG : 'N U T, 0, 0, 0',
	X = 1228.333  mm,	Y = 208.047  mm,	Z = -231.942  mm,
	W = 0.000 deg,	P = 30.000 deg,	R = 167.638 deg
};
P[363]{
   GP1:
	UF : 0, UT : 1,		CONFIG : 'N U T, 0, 0, 0',
	X = 1229.699  mm,	Y = 209.473  mm,	Z = -232.264  mm,
	W = 0.000 deg,	P = 30.000 deg,	R = 171.720 deg
};
P[364]{
   GP1:
	UF : 0, UT : 1,		CONFIG : 'N U T, 0, 0, 0',
	X = 1231.064  mm,	Y = 210.898  mm,	Z = -232.586  mm,
	W = 0.000 deg,	P = 30.000 deg,	R = 175.803 deg
};
P[365]{
   GP1:
	UF : 0, UT : 1,		CONFIG : 'N U T, 0, 0, 0',
	X = 1232.430  mm,	Y = 212.323  mm,	Z = -232.908  mm,
	W = 0.000 deg,	P = 30.000 deg,	R = 179.886 deg
};
P[366]{
   GP1:
	UF : 0, UT : 1,		CONFIG : 'N U T, 0, 0, 0',
	X = 1233.278  mm,	Y = 213.208  mm,	Z = -233.108  mm,
	W = 0.000 deg,	P = 30.000 deg,	R = -179.587 deg
};
P[367]{
   GP1:
	UF : 0, UT : 1,		CONFIG : 'N U T, 0, 0, 0',
	X = 1233.273  mm,	Y = 213.966  mm,	Z = -233.108  mm,
	W = 0.000 deg,	P = 30.000 deg,	R = -179.587 deg
};
P[368]{
   GP1:
	UF : 0, UT : 1,		CONFIG : 'N U T, 0, 0, 0',
	X = 1233.258  mm,	Y = 215.966  mm,	Z = -233.107  mm,
	W = 0.000 deg,	P = 30.000 deg,	R = -179.587 deg
};
P[369]{
   GP1:
	UF : 0, UT : 1,		CONFIG : 'N U T, 0, 0, 0',
	X = 1233.244  mm,	Y = 217.966  mm,	Z = -233.107  mm,
	W = 0.000 deg,	P = 30.000 deg,	R = -179.587 deg
};
P[370]{
   GP1:
	UF : 0, UT : 1,		CONFIG : 'N U T, 0, 0, 0',
	X = 1233.229  mm,	Y = 219.966  mm,	Z = -233.107  mm,
	W = 0.000 deg,	P = 30.000 deg,	R = -179.587 deg
};
P[371]{
   GP1:
	UF : 0, UT : 1,		CONFIG : 'N U T, 0, 0, 0',
	X = 1233.215  mm,	Y = 221.966  mm,	Z = -233.107  mm,
	W = 0.000 deg,	P = 30.000 deg,	R = -179.587 deg
};
P[372]{
   GP1:
	UF : 0, UT : 1,		CONFIG : 'N U T, 0, 0, 0',
	X = 1233.206  mm,	Y = 223.208  mm,	Z = -233.107  mm,
	W = 0.000 deg,	P = 30.000 deg,	R = -179.587 deg
};
/END
